C03644=1220.978,171.514,-54.038,-177.762,5.951,148.395
C03645=1220.983,171.266,-54.017,-177.765,5.949,148.395
C03646=1220.988,171.016,-53.994,-177.767,5.948,148.396
C03647=1220.992,170.767,-53.972,-177.770,5.947,148.396
C03648=1220.997,170.518,-53.950,-177.773,5.945,148.397
C03649=1221.001,170.270,-53.928,-177.775,5.943,148.397
C03650=1221.006,170.020,-53.905,-177.777,5.942,148.397
C03651=1221.011,169.771,-53.883,-177.781,5.941,148.398
C03652=1221.015,169.522,-53.861,-177.783,5.940,148.398
C03653=1221.020,169.273,-53.839,-177.785,5.938,148.399
C03654=1221.025,169.025,-53.816,-177.788,5.936,148.399
C03655=1221.029,168.775,-53.794,-177.791,5.936,148.400
C03656=1221.034,168.527,-53.773,-177.793,5.934,148.400
C03657=1221.038,168.277,-53.751,-177.796,5.932,148.400
C03658=1221.043,168.029,-53.729,-177.798,5.931,148.401
C03659=1221.048,167.779,-53.706,-177.801,5.929,148.401
C03660=1221.053,167.530,-53.685,-177.803,5.928,148.402
C03661=1221.057,167.282,-53.662,-177.806,5.927,148.402
C03662=1221.062,167.033,-53.640,-177.809,5.925,148.403
C03663=1221.066,166.784,-53.618,-177.811,5.924,148.403
C03664=1221.071,166.535,-53.596,-177.814,5.922,148.404
C03665=1221.075,166.286,-53.574,-177.816,5.921,148.404
C03666=1221.081,166.037,-53.552,-177.819,5.920,148.405
C03667=1221.085,165.788,-53.530,-177.822,5.918,148.405
C03668=1221.090,165.539,-53.508,-177.824,5.917,148.405
C03669=1221.094,165.290,-53.486,-177.827,5.915,148.406
C03670=1221.099,165.041,-53.465,-177.829,5.915,148.406
C03671=1221.104,164.792,-53.443,-177.832,5.913,148.407
C03672=1221.108,164.543,-53.421,-177.834,5.911,148.407
C03673=1221.113,164.294,-53.399,-177.837,5.910,148.408
C03674=1221.117,164.045,-53.377,-177.840,5.908,148.408
C03675=1221.122,163.796,-53.355,-177.842,5.907,148.408
C03676=1221.127,163.547,-53.333,-177.844,5.906,148.409
C03677=1221.132,163.298,-53.311,-177.848,5.904,148.409
C03678=1221.137,163.049,-53.289,-177.850,5.903,148.410
C03679=1221.141,162.800,-53.267,-177.852,5.901,148.410
C03680=1221.147,162.551,-53.246,-177.855,5.901,148.411
C03681=1221.151,162.301,-53.224,-177.858,5.899,148.411
C03682=1221.156,162.053,-53.203,-177.860,5.897,148.411
C03683=1221.160,161.803,-53.181,-177.863,5.896,148.412
C03684=1221.165,161.555,-53.159,-177.865,5.895,148.412
C03685=1221.170,161.306,-53.137,-177.868,5.894,148.413
C03686=1221.174,161.057,-53.115,-177.870,5.892,148.413
C03687=1221.179,160.808,-53.094,-177.873,5.891,148.414
C03688=1221.183,160.558,-53.072,-177.876,5.889,148.414
C03689=1221.188,160.310,-53.051,-177.878,5.887,148.415
C03690=1221.193,160.061,-53.029,-177.881,5.887,148.415
C03691=1221.198,159.792,-53.006,-177.883,5.885,148.416
C03692=1221.203,159.523,-52.982,-177.887,5.884,148.416
C03693=1221.209,159.254,-52.959,-177.889,5.883,148.417
C03694=1221.213,158.984,-52.936,-177.892,5.881,148.417
C03695=1221.218,158.735,-52.914,-177.894,5.879,148.417
C03696=1221.222,158.487,-52.892,-177.897,5.878,148.418
C03697=1221.227,158.237,-52.870,-177.900,5.877,148.418
C03698=1221.232,157.988,-52.849,-177.902,5.876,148.419
C03699=1221.237,157.740,-52.827,-177.905,5.874,148.419
C03700=1221.241,157.490,-52.805,-177.908,5.872,148.420
C03701=1221.246,157.241,-52.784,-177.910,5.871,148.420
C03702=1221.251,156.992,-52.763,-177.912,5.870,148.421
C03703=1221.255,156.743,-52.741,-177.915,5.869,148.421
C03704=1221.260,156.494,-52.720,-177.918,5.867,148.422
C03705=1221.265,156.245,-52.699,-177.920,5.866,148.422
C03706=1221.270,155.997,-52.677,-177.923,5.865,148.423
C03707=1221.274,155.747,-52.656,-177.925,5.864,148.423
C03708=1221.279,155.498,-52.634,-177.928,5.862,148.423
C03709=1221.284,155.249,-52.612,-177.930,5.861,148.424
C03710=1221.288,155.000,-52.592,-177.933,5.859,148.424
C03711=1221.293,154.751,-52.570,-177.936,5.858,148.425
C03712=1221.298,154.502,-52.549,-177.938,5.857,148.425
C03713=1221.303,154.253,-52.527,-177.941,5.855,148.426
C03714=1221.307,154.003,-52.506,-177.943,5.854,148.426
C03715=1221.312,153.755,-52.484,-177.946,5.853,148.427
C03716=1221.316,153.506,-52.463,-177.948,5.852,148.427
C03717=1221.321,153.256,-52.442,-177.951,5.850,148.427
C03718=1221.326,153.008,-52.420,-177.954,5.849,148.428
C03719=1221.331,152.758,-52.399,-177.956,5.847,148.428
C03720=1221.335,152.510,-52.378,-177.959,5.847,148.429
C03721=1221.339,152.260,-52.357,-177.961,5.845,148.429
C03722=1221.344,152.012,-52.335,-177.964,5.844,148.430
C03723=1221.350,151.762,-52.314,-177.967,5.843,148.430
C03724=1221.354,151.514,-52.293,-177.969,5.842,148.431
C03725=1221.359,151.265,-52.272,-177.971,5.840,148.431
C03726=1221.363,151.015,-52.251,-177.974,5.839,148.432
C03727=1221.368,150.766,-52.229,-177.977,5.837,148.432
C03728=1221.373,150.517,-52.209,-177.979,5.836,148.433
C03729=1221.378,150.269,-52.187,-177.982,5.835,148.433
C03730=1221.383,150.019,-52.166,-177.984,5.834,148.434
C03731=1221.387,149.770,-52.144,-177.987,5.832,148.434
C03732=1221.391,149.521,-52.124,-177.989,5.831,148.435
C03733=1221.397,149.272,-52.103,-177.992,5.830,148.435
C03734=1221.401,149.023,-52.081,-177.995,5.829,148.436
C03735=1221.406,148.774,-52.061,-177.997,5.827,148.436
C03736=1221.410,148.524,-52.039,-178.000,5.827,148.437
C03737=1221.415,148.276,-52.018,-178.003,5.825,148.437
C03738=1221.420,148.027,-51.997,-178.005,5.824,148.437
C03739=1221.425,147.777,-51.976,-178.008,5.822,148.438
C03740=1221.429,147.529,-51.955,-178.010,5.821,148.438
C03741=1221.434,147.280,-51.934,-178.013,5.819,148.439
C03742=1221.439,147.030,-51.913,-178.015,5.819,148.439
C03743=1221.443,146.781,-51.892,-178.018,5.817,148.440
C03744=1221.448,146.532,-51.871,-178.020,5.816,148.440
C03745=1221.453,146.283,-51.850,-178.023,5.815,148.441
C03746=1221.458,146.034,-51.829,-178.025,5.814,148.441
C03747=1221.463,145.785,-51.808,-178.028,5.812,148.442
C03748=1221.467,145.536,-51.787,-178.031,5.811,148.442
C03749=1221.472,145.286,-51.766,-178.034,5.810,148.443
C03750=1221.476,145.037,-51.746,-178.036,5.809,148.443
C03751=1221.481,144.788,-51.725,-178.038,5.807,148.443
C03752=1221.486,144.540,-51.703,-178.041,5.806,148.444
C03753=1221.491,144.291,-51.683,-178.044,5.804,148.444
C03754=1221.496,144.041,-51.662,-178.046,5.804,148.445
C03755=1221.500,143.792,-51.641,-178.049,5.802,148.446
C03756=1221.505,143.543,-51.620,-178.051,5.801,148.446
C03757=1221.510,143.294,-51.600,-178.054,5.800,148.447
C03758=1221.514,143.045,-51.578,-178.056,5.799,148.447
C03759=1221.519,142.796,-51.558,-178.059,5.798,148.448
C03760=1221.524,142.547,-51.537,-178.062,5.796,148.448
C03761=1221.528,142.298,-51.516,-178.064,5.795,148.449
C03762=1221.533,142.048,-51.495,-178.067,5.794,148.449
C03763=1221.538,141.799,-51.475,-178.069,5.793,148.449
C03764=1221.543,141.550,-51.454,-178.072,5.791,148.450
C03765=1221.547,141.301,-51.434,-178.074,5.790,148.450
C03766=1221.553,141.052,-51.413,-178.077,5.789,148.451
C03767=1221.557,140.803,-51.392,-178.080,5.788,148.451
C03768=1221.562,140.554,-51.371,-178.083,5.786,148.452
C03769=1221.567,140.305,-51.351,-178.085,5.785,148.452
C03770=1221.571,140.056,-51.330,-178.087,5.784,148.453
C03771=1221.576,139.807,-51.310,-178.090,5.783,148.453
C03772=1221.581,139.558,-51.289,-178.092,5.782,148.454
C03773=1221.586,139.308,-51.268,-178.095,5.781,148.454
C03774=1221.590,139.059,-51.248,-178.097,5.780,148.455
C03775=1221.595,138.810,-51.227,-178.101,5.778,148.455
C03776=1221.600,138.561,-51.206,-178.103,5.777,148.456
C03777=1221.604,138.312,-51.186,-178.105,5.775,148.456
C03778=1221.609,138.063,-51.165,-178.108,5.775,148.457
C03779=1221.614,137.814,-51.145,-178.110,5.774,148.457
C03780=1221.618,137.565,-51.124,-178.113,5.772,148.458
C03781=1221.623,137.316,-51.103,-178.115,5.771,148.458
C03782=1221.628,137.067,-51.083,-178.119,5.770,148.459
C03783=1221.633,136.818,-51.062,-178.121,5.769,148.459
C03784=1221.638,136.569,-51.042,-178.124,5.767,148.460
C03785=1221.642,136.320,-51.021,-178.126,5.766,148.460
C03786=1221.647,136.070,-51.001,-178.128,5.765,148.461
C03787=1221.652,135.821,-50.981,-178.131,5.764,148.461
C03788=1221.656,135.572,-50.960,-178.133,5.763,148.462
C03789=1221.662,135.323,-50.939,-178.137,5.762,148.462
C03790=1221.666,135.074,-50.919,-178.139,5.761,148.463
C03791=1221.670,134.825,-50.899,-178.141,5.760,148.463
C03792=1221.675,134.575,-50.879,-178.144,5.758,148.464
C03793=1221.680,134.326,-50.858,-178.146,5.757,148.464
C03794=1221.685,134.077,-50.838,-178.149,5.756,148.465
C03795=1221.690,133.808,-50.816,-178.152,5.755,148.465
C03796=1221.695,133.540,-50.794,-178.154,5.753,148.466
C03797=1221.700,133.271,-50.771,-178.157,5.753,148.466
C03798=1221.705,133.002,-50.750,-178.160,5.751,148.467
C03799=1221.710,132.753,-50.729,-178.162,5.750,148.467
C03800=1221.714,132.504,-50.709,-178.165,5.749,148.468
C03801=1221.720,132.255,-50.690,-178.168,5.748,148.468
C03802=1221.725,132.006,-50.669,-178.171,5.746,148.469
C03803=1221.729,131.757,-50.648,-178.173,5.745,148.469
C03804=1221.734,131.508,-50.629,-178.175,5.745,148.470
C03805=1221.738,131.259,-50.608,-178.178,5.743,148.470
C03806=1221.743,131.010,-50.588,-178.181,5.742,148.471
C03807=1221.748,130.760,-50.568,-178.183,5.740,148.471
C03808=1221.753,130.511,-50.547,-178.186,5.740,148.472
C03809=1221.757,130.262,-50.527,-178.188,5.739,148.472
C03810=1221.763,130.013,-50.508,-178.191,5.737,148.473
C03811=1221.767,129.764,-50.487,-178.193,5.736,148.473
C03812=1221.772,129.514,-50.467,-178.197,5.735,148.474
C03813=1221.777,129.265,-50.447,-178.199,5.734,148.474
C03814=1221.781,129.016,-50.426,-178.201,5.733,148.475
C03815=1221.786,128.767,-50.407,-178.204,5.732,148.476
C03816=1221.791,128.518,-50.386,-178.207,5.731,148.476
C03817=1221.796,128.269,-50.367,-178.209,5.730,148.477
C03818=1221.800,128.020,-50.347,-178.212,5.729,148.477
C03819=1221.805,127.771,-50.326,-178.214,5.728,148.478
C03820=1221.810,127.521,-50.306,-178.217,5.726,148.478
C03821=1221.815,127.272,-50.286,-178.219,5.725,148.479
C03822=1221.819,127.023,-50.266,-178.222,5.725,148.479
C03823=1221.824,126.774,-50.246,-178.225,5.723,148.480
C03824=1221.829,126.525,-50.226,-178.227,5.722,148.480
C03825=1221.834,126.276,-50.206,-178.229,5.721,148.481
C03826=1221.838,126.026,-50.186,-178.232,5.720,148.481
C03827=1221.843,125.777,-50.166,-178.235,5.719,148.482
C03828=1221.848,125.528,-50.147,-178.237,5.718,148.482
C03829=1221.853,125.279,-50.127,-178.240,5.716,148.483
C03830=1221.857,125.030,-50.107,-178.242,5.716,148.483
C03831=1221.862,124.780,-50.087,-178.245,5.714,148.484
C03832=1221.866,124.531,-50.067,-178.248,5.713,148.484
C03833=1221.872,124.283,-50.047,-178.250,5.712,148.485
C03834=1221.876,124.034,-50.027,-178.253,5.711,148.485
C03835=1221.881,123.784,-50.007,-178.255,5.710,148.486
C03836=1221.886,123.534,-49.988,-178.258,5.709,148.486
C03837=1221.891,123.286,-49.968,-178.260,5.707,148.487
C03838=1221.896,123.037,-49.948,-178.263,5.707,148.487
C03839=1221.900,122.787,-49.928,-178.265,5.706,148.488
C03840=1221.905,122.538,-49.908,-178.268,5.704,148.489
C03841=1221.910,122.289,-49.889,-178.270,5.703,148.489
C03842=1221.915,122.040,-49.869,-178.273,5.703,148.490
C03843=1221.919,121.791,-49.849,-178.276,5.701,148.490
C03844=1221.924,121.541,-49.829,-178.278,5.700,148.491
C03845=1221.929,121.292,-49.810,-178.281,5.700,148.491
C03846=1221.934,121.043,-49.789,-178.284,5.698,148.492
C03847=1221.939,120.794,-49.770,-178.286,5.697,148.492
C03848=1221.944,120.545,-49.750,-178.288,5.696,148.493
C03849=1221.948,120.296,-49.730,-178.292,5.695,148.493
C03850=1221.953,120.046,-49.710,-178.294,5.694,148.494
C03851=1221.958,119.797,-49.691,-178.296,5.693,148.494
C03852=1221.963,119.548,-49.671,-178.299,5.692,148.495
C03853=1221.968,119.298,-49.652,-178.302,5.691,148.495
C03854=1221.972,119.050,-49.632,-178.304,5.690,148.496
C03855=1221.977,118.801,-49.613,-178.307,5.689,148.496
C03856=1221.982,118.551,-49.593,-178.309,5.688,148.497
C03857=1221.986,118.302,-49.573,-178.312,5.687,148.497
C03858=1221.992,118.053,-49.554,-178.315,5.686,148.498
C03859=1221.996,117.804,-49.534,-178.317,5.685,148.498
C03860=1222.001,117.554,-49.514,-178.320,5.684,148.499
C03861=1222.006,117.306,-49.495,-178.322,5.682,148.500
C03862=1222.010,117.056,-49.476,-178.325,5.682,148.500
C03863=1222.015,116.807,-49.456,-178.327,5.681,148.501
C03864=1222.020,116.558,-49.437,-178.330,5.680,148.501
C03865=1222.025,116.308,-49.417,-178.333,5.679,148.502
C03866=1222.030,116.059,-49.397,-178.335,5.678,148.502
C03867=1222.034,115.811,-49.378,-178.337,5.677,148.503
C03868=1222.039,115.561,-49.358,-178.340,5.675,148.503
C03869=1222.044,115.312,-49.339,-178.343,5.675,148.504
C03870=1222.049,115.063,-49.319,-178.345,5.674,148.504
C03871=1222.054,114.813,-49.300,-178.348,5.672,148.505
C03872=1222.058,114.565,-49.281,-178.351,5.672,148.506
C03873=1222.063,114.315,-49.261,-178.353,5.671,148.506
C03874=1222.068,114.065,-49.242,-178.355,5.670,148.507
C03875=1222.073,113.817,-49.222,-178.358,5.668,148.507
C03876=1222.077,113.567,-49.203,-178.361,5.668,148.508
C03877=1222.083,113.319,-49.184,-178.363,5.667,148.508
C03878=1222.087,113.069,-49.164,-178.366,5.665,148.509
C03879=1222.092,112.819,-49.145,-178.369,5.665,148.509
C03880=1222.097,112.571,-49.126,-178.371,5.664,148.510
C03881=1222.101,112.321,-49.106,-178.373,5.663,148.510
C03882=1222.107,112.072,-49.087,-178.376,5.661,148.511
C03883=1222.111,111.823,-49.067,-178.379,5.661,148.511
C03884=1222.116,111.574,-49.049,-178.381,5.660,148.512
C03885=1222.121,111.325,-49.029,-178.384,5.658,148.512
C03886=1222.126,111.075,-49.009,-178.387,5.658,148.513
C03887=1222.130,110.827,-48.991,-178.389,5.657,148.514
C03888=1222.135,110.577,-48.971,-178.391,5.656,148.514
C03889=1222.141,110.327,-48.952,-178.394,5.654,148.515
C03890=1222.145,110.078,-48.933,-178.397,5.654,148.515
C03891=1222.150,109.829,-48.914,-178.399,5.653,148.516
C03892=1222.155,109.580,-48.894,-178.401,5.652,148.516
C03893=1222.159,109.331,-48.876,-178.404,5.651,148.517
C03894=1222.164,109.082,-48.856,-178.407,5.650,148.517
C03895=1222.169,108.833,-48.837,-178.409,5.649,148.518
C03896=1222.174,108.583,-48.818,-178.412,5.648,148.519
C03897=1222.179,108.334,-48.799,-178.415,5.647,148.519
C03898=1222.183,108.085,-48.780,-178.417,5.646,148.520
C03899=1222.188,107.817,-48.759,-178.420,5.645,148.520
C03900=1222.194,107.548,-48.739,-178.422,5.644,148.521
C03901=1222.199,107.280,-48.718,-178.425,5.643,148.521
C03902=1222.204,107.011,-48.697,-178.428,5.642,148.522
C03903=1222.209,106.762,-48.679,-178.431,5.641,148.523
C03904=1222.214,106.512,-48.660,-178.433,5.640,148.523
C03905=1222.218,106.264,-48.641,-178.436,5.639,148.524
C03906=1222.223,106.014,-48.621,-178.439,5.638,148.524
C03907=1222.228,105.765,-48.603,-178.441,5.637,148.525
C03908=1222.233,105.515,-48.584,-178.443,5.636,148.525
C03909=1222.238,105.267,-48.564,-178.446,5.635,148.526
C03910=1222.242,105.017,-48.545,-178.449,5.634,148.526
C03911=1222.248,104.768,-48.527,-178.451,5.633,148.527
C03912=1222.252,104.519,-48.508,-178.454,5.632,148.527
C03913=1222.257,104.270,-48.488,-178.456,5.632,148.528
C03914=1222.261,104.020,-48.470,-178.459,5.630,148.529
C03915=1222.267,103.771,-48.451,-178.461,5.629,148.529
C03916=1222.271,103.522,-48.432,-178.464,5.629,148.530
C03917=1222.276,103.272,-48.413,-178.466,5.628,148.530
C03918=1222.281,103.024,-48.394,-178.469,5.626,148.531
C03919=1222.286,102.773,-48.375,-178.472,5.626,148.532
C03920=1222.291,102.525,-48.357,-178.474,5.625,148.532
C03921=1222.295,102.275,-48.337,-178.477,5.624,148.533
C03922=1222.300,102.026,-48.319,-178.479,5.624,148.533
C03923=1222.305,101.778,-48.300,-178.482,5.622,148.534
C03924=1222.310,101.527,-48.281,-178.485,5.621,148.534
C03925=1222.315,101.279,-48.263,-178.487,5.620,148.535
C03926=1222.320,101.029,-48.244,-178.489,5.620,148.535
C03927=1222.324,100.780,-48.225,-178.493,5.618,148.536
C03928=1222.330,100.531,-48.206,-178.495,5.617,148.536
C03929=1222.334,100.281,-48.187,-178.497,5.617,148.537
C03930=1222.339,100.033,-48.169,-178.500,5.616,148.538
C03931=1222.344,99.783,-48.150,-178.502,5.615,148.538
C03932=1222.348,99.534,-48.131,-178.505,5.614,148.539
C03933=1222.354,99.285,-48.113,-178.508,5.613,148.539
C03934=1222.358,99.035,-48.094,-178.510,5.612,148.540
C03935=1222.363,98.786,-48.076,-178.513,5.612,148.540
C03936=1222.368,98.537,-48.057,-178.515,5.611,148.541
C03937=1222.372,98.287,-48.038,-178.518,5.609,148.542
C03938=1222.377,98.038,-48.020,-178.521,5.609,148.542
C03939=1222.383,97.789,-48.001,-178.523,5.608,148.543
C03940=1222.387,97.539,-47.982,-178.525,5.607,148.543
C03941=1222.392,97.291,-47.964,-178.528,5.606,148.544
C03942=1222.397,97.041,-47.945,-178.531,5.605,148.545
C03943=1222.402,96.792,-47.927,-178.533,5.604,148.545
C03944=1222.406,96.543,-47.908,-178.536,5.604,148.546
C03945=1222.412,96.293,-47.889,-178.538,5.603,148.546
C03946=1222.416,96.044,-47.870,-178.541,5.602,148.547
C03947=1222.421,95.795,-47.852,-178.544,5.601,148.547
C03948=1222.426,95.546,-47.834,-178.546,5.600,148.548
C03949=1222.430,95.296,-47.815,-178.549,5.599,148.548
C03950=1222.435,95.047,-47.797,-178.551,5.598,148.549
C03951=1222.441,94.798,-47.778,-178.554,5.598,148.550
C03952=1222.445,94.548,-47.759,-178.556,5.596,148.550
C03953=1222.450,94.299,-47.741,-178.559,5.595,148.551
C03954=1222.455,94.050,-47.723,-178.562,5.595,148.551
C03955=1222.460,93.801,-47.704,-178.564,5.594,148.552
C03956=1222.464,93.551,-47.686,-178.566,5.593,148.552
C03957=1222.469,93.302,-47.668,-178.569,5.593,148.553
C03958=1222.474,93.053,-47.650,-178.572,5.591,148.553
C03959=1222.480,92.804,-47.630,-178.574,5.590,148.554
C03960=1222.484,92.554,-47.612,-178.577,5.590,148.555
C03961=1222.489,92.305,-47.594,-178.579,5.589,148.555
C03962=1222.494,92.056,-47.576,-178.582,5.588,148.556
C03963=1222.498,91.807,-47.557,-178.585,5.587,148.557
C03964=1222.503,91.557,-47.538,-178.587,5.586,148.557
C03965=1222.508,91.308,-47.520,-178.590,5.585,148.558
C03966=1222.513,91.059,-47.502,-178.592,5.585,148.558
C03967=1222.518,90.810,-47.484,-178.594,5.584,148.559
C03968=1222.522,90.560,-47.466,-178.597,5.583,148.559
C03969=1222.527,90.311,-47.447,-178.600,5.582,148.560
C03970=1222.533,90.062,-47.429,-178.602,5.581,148.560
C03971=1222.538,89.812,-47.411,-178.605,5.580,148.561
C03972=1222.542,89.563,-47.392,-178.608,5.580,148.562
C03973=1222.547,89.313,-47.374,-178.610,5.579,148.562
C03974=1222.552,89.064,-47.356,-178.612,5.578,148.563
C03975=1222.557,88.815,-47.339,-178.615,5.577,148.563
C03976=1222.561,88.567,-47.320,-178.618,5.576,148.564
C03977=1222.566,88.316,-47.301,-178.620,5.575,148.564
C03978=1222.571,88.067,-47.283,-178.623,5.574,148.565
C03979=1222.576,87.818,-47.265,-178.626,5.574,148.566
C03980=1222.581,87.569,-47.247,-178.628,5.573,148.566
C03981=1222.586,87.320,-47.229,-178.630,5.572,148.567
C03982=1222.590,87.070,-47.211,-178.633,5.572,148.568
C03983=1222.595,86.821,-47.193,-178.636,5.570,148.568
C03984=1222.600,86.571,-47.175,-178.638,5.569,148.569
C03985=1222.605,86.322,-47.157,-178.641,5.569,148.569
C03986=1222.610,86.073,-47.139,-178.644,5.568,148.570
C03987=1222.615,85.824,-47.121,-178.646,5.567,148.570
C03988=1222.619,85.574,-47.102,-178.648,5.567,148.571
C03989=1222.624,85.325,-47.084,-178.651,5.566,148.572
C03990=1222.629,85.076,-47.066,-178.654,5.565,148.572
C03991=1222.635,84.826,-47.048,-178.656,5.564,148.573
C03992=1222.640,84.577,-47.030,-178.659,5.563,148.573
C03993=1222.644,84.328,-47.012,-178.661,5.562,148.574
C03994=1222.649,84.079,-46.994,-178.664,5.562,148.574
C03995=1222.654,83.829,-46.976,-178.666,5.561,148.575
C03996=1222.659,83.580,-46.958,-178.669,5.560,148.576
C03997=1222.663,83.330,-46.940,-178.671,5.560,148.576
C03998=1222.668,83.081,-46.922,-178.674,5.558,148.577
C03999=1222.674,82.831,-46.904,-178.677,5.557,148.577
C04000=1222.679,82.582,-46.886,-178.679,5.557,148.578
C04001=1222.683,82.333,-46.869,-178.682,5.556,148.579
C04002=1222.688,82.084,-46.851,-178.684,5.555,148.579
C04003=1222.693,81.816,-46.831,-178.687,5.555,148.580
C04004=1222.699,81.547,-46.812,-178.690,5.553,148.580
C04005=1222.704,81.279,-46.793,-178.693,5.553,148.581
C04006=1222.709,81.010,-46.773,-178.695,5.552,148.582
C04007=1222.714,80.761,-46.755,-178.698,5.552,148.582
C04008=1222.719,80.512,-46.738,-178.700,5.551,148.583
C04009=1222.723,80.263,-46.720,-178.703,5.549,148.584
C04010=1222.728,80.013,-46.703,-178.706,5.549,148.584
C04011=1222.733,79.764,-46.685,-178.708,5.548,148.585
C04012=1222.738,79.515,-46.667,-178.711,5.547,148.585
C04013=1222.743,79.266,-46.649,-178.713,5.546,148.586
C04014=1222.748,79.016,-46.632,-178.716,5.546,148.587
C04015=1222.753,78.767,-46.614,-178.718,5.545,148.587
C04016=1222.757,78.517,-46.595,-178.721,5.544,148.588
C04017=1222.762,78.268,-46.577,-178.723,5.544,148.588
C04018=1222.767,78.018,-46.561,-178.726,5.543,148.589
C04019=1222.772,77.769,-46.543,-178.729,5.542,148.590
C04020=1222.777,77.520,-46.525,-178.731,5.541,148.590
C04021=1222.781,77.271,-46.507,-178.734,5.540,148.591
C04022=1222.787,77.021,-46.489,-178.736,5.540,148.591
C04023=1222.792,76.772,-46.471,-178.739,5.539,148.592
C04024=1222.796,76.523,-46.454,-178.741,5.538,148.592
C04025=1222.801,76.273,-46.437,-178.744,5.538,148.593
C04026=1222.806,76.024,-46.419,-178.746,5.537,148.594
C04027=1222.811,75.775,-46.401,-178.749,5.536,148.594
C04028=1222.816,75.525,-46.384,-178.751,5.535,148.595
C04029=1222.821,75.276,-46.366,-178.754,5.535,148.596
C04030=1222.825,75.027,-46.348,-178.756,5.534,148.596
C04031=1222.830,74.777,-46.331,-178.760,5.533,148.597
C04032=1222.835,74.528,-46.313,-178.762,5.532,148.597
C04033=1222.840,74.278,-46.296,-178.764,5.531,148.598
C04034=1222.845,74.029,-46.278,-178.767,5.531,148.599
C04035=1222.850,73.780,-46.260,-178.770,5.530,148.599
C04036=1222.855,73.530,-46.243,-178.772,5.529,148.600
C04037=1222.860,73.282,-46.226,-178.774,5.529,148.600
C04038=1222.865,73.032,-46.209,-178.777,5.528,148.601
C04039=1222.870,72.783,-46.191,-178.780,5.528,148.602
C04040=1222.875,72.533,-46.174,-178.782,5.527,148.602
C04041=1222.880,72.284,-46.156,-178.784,5.526,148.603
C04042=1222.884,72.035,-46.139,-178.787,5.525,148.603
C04043=1222.889,71.786,-46.121,-178.790,5.525,148.604
C04044=1222.894,71.536,-46.104,-178.792,5.524,148.605
C04045=1222.899,71.287,-46.086,-178.795,5.523,148.605
C04046=1222.904,71.037,-46.069,-178.798,5.522,148.606
C04047=1222.909,70.788,-46.051,-178.800,5.521,148.606
C04048=1222.914,70.538,-46.034,-178.803,5.521,148.607
C04049=1222.918,70.289,-46.016,-178.806,5.520,148.608
C04050=1222.923,70.039,-45.999,-178.808,5.519,148.608
C04051=1222.929,69.791,-45.982,-178.810,5.519,148.609
C04052=1222.933,69.541,-45.965,-178.813,5.518,148.610
C04053=1222.939,69.292,-45.948,-178.816,5.518,148.610
C04054=1222.943,69.043,-45.930,-178.818,5.517,148.611
C04055=1222.948,68.793,-45.913,-178.820,5.516,148.611
C04056=1222.953,68.544,-45.895,-178.823,5.515,148.612
C04057=1222.957,68.294,-45.878,-178.826,5.515,148.613
C04058=1222.963,68.045,-45.861,-178.828,5.514,148.613
C04059=1222.967,67.795,-45.843,-178.830,5.513,148.614
C04060=1222.973,67.547,-45.827,-178.833,5.513,148.614
C04061=1222.977,67.297,-45.809,-178.836,5.512,148.615
C04062=1222.982,67.048,-45.792,-178.838,5.512,148.616
C04063=1222.987,66.798,-45.775,-178.841,5.511,148.616
C04064=1222.992,66.549,-45.757,-178.843,5.510,148.617
C04065=1222.997,66.299,-45.740,-178.846,5.509,148.617
C04066=1223.002,66.050,-45.723,-178.849,5.508,148.618
C04067=1223.007,65.802,-45.706,-178.852,5.508,148.619
C04068=1223.012,65.552,-45.689,-178.854,5.507,148.619
C04069=1223.016,65.302,-45.672,-178.856,5.506,148.620
C04070=1223.021,65.052,-45.655,-178.859,5.505,148.621
C04071=1223.026,64.804,-45.637,-178.862,5.505,148.621
C04072=1223.031,64.554,-45.620,-178.864,5.504,148.622
C04073=1223.037,64.305,-45.603,-178.867,5.504,148.623
C04074=1223.041,64.055,-45.587,-178.869,5.503,148.623
C04075=1223.046,63.806,-45.569,-178.872,5.502,148.624
C04076=1223.051,63.557,-45.552,-178.874,5.502,148.624
C04077=1223.056,63.307,-45.535,-178.877,5.501,148.625
C04078=1223.060,63.057,-45.518,-178.879,5.501,148.626
C04079=1223.066,62.809,-45.500,-178.882,5.500,148.626
C04080=1223.070,62.559,-45.484,-178.884,5.499,148.627
C04081=1223.075,62.310,-45.466,-178.887,5.498,148.627
C04082=1223.080,62.060,-45.450,-178.890,5.498,148.628
C04083=1223.086,61.811,-45.433,-178.892,5.497,148.629
C04084=1223.090,61.561,-45.416,-178.894,5.496,148.629
C04085=1223.094,61.313,-45.399,-178.897,5.496,148.630
C04086=1223.100,61.063,-45.381,-178.900,5.495,148.630
C04087=1223.104,60.813,-45.365,-178.902,5.495,148.631
C04088=1223.110,60.564,-45.348,-178.905,5.494,148.632
C04089=1223.114,60.315,-45.331,-178.907,5.493,148.632
C04090=1223.120,60.065,-45.314,-178.910,5.493,148.633
C04091=1223.124,59.815,-45.297,-178.912,5.492,148.634
C04092=1223.130,59.566,-45.280,-178.915,5.491,148.634
C04093=1223.134,59.317,-45.264,-178.917,5.491,148.635
C04094=1223.139,59.068,-45.246,-178.920,5.490,148.636
C04095=1223.144,58.818,-45.229,-178.922,5.489,148.636
C04096=1223.149,58.569,-45.213,-178.925,5.489,148.637
C04097=1223.154,58.320,-45.196,-178.928,5.488,148.637
C04098=1223.159,58.070,-45.179,-178.930,5.488,148.638
C04099=1223.164,57.821,-45.163,-178.933,5.487,148.639
C04100=1223.169,57.572,-45.145,-178.935,5.487,148.639
C04101=1223.173,57.322,-45.129,-178.938,5.486,148.640
C04102=1223.178,57.073,-45.112,-178.940,5.485,148.640
C04103=1223.184,56.824,-45.095,-178.943,5.484,148.641
C04104=1223.188,56.574,-45.078,-178.945,5.484,148.642
C04105=1223.193,56.325,-45.062,-178.948,5.483,148.642
C04106=1223.198,56.075,-45.045,-178.950,5.482,148.643
C04107=1223.203,55.807,-45.027,-178.953,5.482,148.644
C04108=1223.209,55.538,-45.009,-178.956,5.482,148.644
C04109=1223.214,55.270,-44.991,-178.959,5.481,148.645
C04110=1223.219,55.002,-44.973,-178.962,5.480,148.646
C04111=1223.225,54.752,-44.956,-178.965,5.479,148.646
C04112=1223.229,54.502,-44.939,-178.967,5.478,148.647
C04113=1223.234,54.254,-44.923,-178.969,5.478,148.648
C04114=1223.239,54.004,-44.906,-178.971,5.478,148.648
C04115=1223.244,53.754,-44.890,-178.974,5.477,148.649
C04116=1223.249,53.505,-44.874,-178.977,5.477,148.650
C04117=1223.254,53.255,-44.857,-178.979,5.476,148.650
C04118=1223.259,53.006,-44.840,-178.981,5.475,148.651
C04119=1223.264,52.757,-44.823,-178.984,5.475,148.651
C04120=1223.268,52.507,-44.807,-178.987,5.474,148.652
C04121=1223.273,52.259,-44.790,-178.989,5.474,148.653
C04122=1223.279,52.008,-44.774,-178.992,5.473,148.653
C04123=1223.283,51.759,-44.757,-178.995,5.472,148.654
C04124=1223.289,51.510,-44.741,-178.997,5.472,148.654
C04125=1223.293,51.260,-44.724,-178.999,5.471,148.655
C04126=1223.298,51.011,-44.707,-179.002,5.470,148.656
C04127=1223.303,50.762,-44.691,-179.005,5.470,148.656
C04128=1223.308,50.512,-44.675,-179.007,5.469,148.657
C04129=1223.313,50.263,-44.658,-179.010,5.469,148.658
C04130=1223.318,50.014,-44.642,-179.013,5.468,148.658
C04131=1223.322,49.764,-44.625,-179.015,5.467,148.659
C04132=1223.328,49.514,-44.609,-179.017,5.467,148.660
C04133=1223.333,49.265,-44.592,-179.020,5.466,148.660
C04134=1223.338,49.016,-44.576,-179.023,5.466,148.661
C04135=1223.342,48.767,-44.559,-179.025,5.465,148.662
C04136=1223.347,48.516,-44.543,-179.028,5.464,148.662
C04137=1223.352,48.268,-44.527,-179.031,5.464,148.663
C04138=1223.357,48.018,-44.510,-179.033,5.463,148.663
C04139=1223.363,47.768,-44.494,-179.035,5.462,148.664
C04140=1223.367,47.519,-44.477,-179.037,5.463,148.665
C04141=1223.372,47.270,-44.461,-179.040,5.462,148.665
C04142=1223.377,47.020,-44.445,-179.043,5.461,148.666
C04143=1223.382,46.771,-44.429,-179.045,5.461,148.667
C04144=1223.387,46.522,-44.412,-179.048,5.460,148.667
C04145=1223.392,46.272,-44.396,-179.051,5.460,148.668
C04146=1223.397,46.023,-44.379,-179.053,5.459,148.669
C04147=1223.402,45.773,-44.363,-179.055,5.458,148.669
C04148=1223.407,45.524,-44.347,-179.058,5.458,148.670
C04149=1223.412,45.274,-44.330,-179.061,5.457,148.671
C04150=1223.417,45.025,-44.315,-179.063,5.457,148.671
C04151=1223.422,44.775,-44.298,-179.066,5.456,148.672
C04152=1223.427,44.527,-44.282,-179.069,5.456,148.673
C04153=1223.431,44.276,-44.266,-179.071,5.455,148.673
C04154=1223.436,44.028,-44.250,-179.073,5.454,148.674
C04155=1223.441,43.778,-44.234,-179.076,5.454,148.674
C04156=1223.446,43.529,-44.217,-179.078,5.454,148.675
C04157=1223.451,43.279,-44.201,-179.081,5.453,148.676
C04158=1223.456,43.030,-44.185,-179.083,5.453,148.676
C04159=1223.461,42.780,-44.168,-179.086,5.452,148.677
C04160=1223.466,42.531,-44.153,-179.089,5.452,148.678
C04161=1223.471,42.282,-44.136,-179.091,5.451,148.678
C04162=1223.476,42.032,-44.121,-179.093,5.450,148.679
C04163=1223.480,41.783,-44.104,-179.096,5.450,148.679
C04164=1223.486,41.533,-44.088,-179.099,5.449,148.680
C04165=1223.491,41.283,-44.072,-179.101,5.448,148.681
C04166=1223.496,41.034,-44.056,-179.104,5.448,148.682
C04167=1223.500,40.784,-44.040,-179.107,5.447,148.682
C04168=1223.506,40.536,-44.024,-179.109,5.447,148.683
C04169=1223.511,40.286,-44.008,-179.111,5.447,148.684
C04170=1223.515,40.037,-43.991,-179.113,5.446,148.684
C04171=1223.521,39.787,-43.976,-179.116,5.446,148.685
C04172=1223.525,39.538,-43.959,-179.119,5.445,148.685
C04173=1223.531,39.288,-43.944,-179.121,5.444,148.686
C04174=1223.535,39.038,-43.928,-179.124,5.444,148.687
C04175=1223.541,38.789,-43.911,-179.127,5.443,148.687
C04176=1223.545,38.539,-43.895,-179.129,5.443,148.688
C04177=1223.550,38.291,-43.879,-179.132,5.442,148.689
C04178=1223.556,38.041,-43.864,-179.135,5.442,148.689
C04179=1223.561,37.791,-43.848,-179.137,5.441,148.690
C04180=1223.566,37.542,-43.831,-179.139,5.441,148.691
C04181=1223.570,37.292,-43.815,-179.141,5.440,148.691
C04182=1223.575,37.043,-43.800,-179.144,5.440,148.692
C04183=1223.580,36.794,-43.784,-179.147,5.439,148.693
C04184=1223.585,36.544,-43.768,-179.149,5.439,148.693
C04185=1223.590,36.295,-43.752,-179.152,5.438,148.694
C04186=1223.595,36.045,-43.736,-179.155,5.438,148.695
C04187=1223.600,35.796,-43.720,-179.157,5.437,148.695
C04188=1223.606,35.546,-43.705,-179.159,5.436,148.696
C04189=1223.610,35.297,-43.689,-179.162,5.436,148.696
C04190=1223.615,35.048,-43.673,-179.164,5.436,148.697
C04191=1223.620,34.799,-43.657,-179.167,5.435,148.698
C04192=1223.625,34.548,-43.641,-179.169,5.435,148.698
C04193=1223.630,34.299,-43.626,-179.172,5.434,148.699
C04194=1223.635,34.050,-43.609,-179.175,5.434,148.700
C04195=1223.639,33.800,-43.594,-179.177,5.433,148.700
C04196=1223.645,33.551,-43.579,-179.180,5.433,148.701
C04197=1223.650,33.301,-43.563,-179.183,5.432,148.702
C04198=1223.655,33.052,-43.546,-179.184,5.432,148.702
C04199=1223.660,32.803,-43.531,-179.187,5.431,148.703
C04200=1223.664,32.553,-43.515,-179.189,5.431,148.704
C04201=1223.670,32.304,-43.500,-179.192,5.430,148.704
C04202=1223.675,32.054,-43.484,-179.195,5.430,148.705
C04203=1223.680,31.804,-43.468,-179.197,5.429,148.706
C04204=1223.685,31.555,-43.452,-179.200,5.429,148.706
C04205=1223.689,31.306,-43.437,-179.203,5.428,148.707
C04206=1223.694,31.056,-43.421,-179.205,5.428,148.708
C04207=1223.700,30.807,-43.405,-179.207,5.428,148.708
C04208=1223.705,30.557,-43.390,-179.210,5.427,148.709
C04209=1223.710,30.308,-43.375,-179.212,5.426,148.709
C04210=1223.714,30.058,-43.359,-179.215,5.426,148.710
C04211=1223.720,29.790,-43.342,-179.218,5.426,148.711
C04212=1223.726,29.521,-43.325,-179.221,5.425,148.712
C04213=1223.730,29.253,-43.308,-179.223,5.425,148.712
C04214=1223.736,28.984,-43.291,-179.226,5.424,148.713
C04215=1223.741,28.734,-43.275,-179.229,5.424,148.714
C04216=1223.745,28.485,-43.260,-179.231,5.423,148.714
C04217=1223.751,28.236,-43.245,-179.234,5.422,148.715
C04218=1223.756,27.986,-43.229,-179.236,5.423,148.716
C04219=1223.761,27.736,-43.213,-179.239,5.422,148.716
C04220=1223.766,27.487,-43.198,-179.241,5.421,148.717
C04221=1223.771,27.238,-43.183,-179.243,5.421,148.718
C04222=1223.776,26.988,-43.167,-179.246,5.420,148.718
C04223=1223.780,26.739,-43.152,-179.249,5.420,148.719
C04224=1223.786,26.489,-43.136,-179.251,5.419,148.720
C04225=1223.791,26.240,-43.121,-179.253,5.419,148.720
C04226=1223.796,25.991,-43.106,-179.256,5.419,148.721
C04227=1223.801,25.741,-43.090,-179.259,5.418,148.722
C04228=1223.805,25.492,-43.075,-179.261,5.418,148.722
C04229=1223.811,25.242,-43.059,-179.264,5.417,148.723
C04230=1223.816,24.993,-43.044,-179.267,5.417,148.724
C04231=1223.820,24.743,-43.028,-179.269,5.416,148.724
C04232=1223.826,24.493,-43.013,-179.271,5.416,148.725
C04233=1223.830,24.244,-42.998,-179.274,5.416,148.726
C04234=1223.836,23.994,-42.983,-179.276,5.415,148.726
C04235=1223.841,23.745,-42.967,-179.279,5.414,148.727
C04236=1223.845,23.495,-42.952,-179.281,5.414,148.728
C04237=1223.851,23.246,-42.936,-179.284,5.413,148.728
C04238=1223.855,22.997,-42.921,-179.286,5.414,148.729
C04239=1223.861,22.747,-42.906,-179.289,5.413,148.730
C04240=1223.865,22.498,-42.891,-179.291,5.413,148.730
C04241=1223.870,22.248,-42.875,-179.294,5.412,148.731
C04242=1223.876,21.998,-42.860,-179.297,5.411,148.732
C04243=1223.880,21.749,-42.845,-179.299,5.411,148.732
C04244=1223.886,21.500,-42.829,-179.301,5.411,148.733
C04245=1223.890,21.251,-42.814,-179.304,5.411,148.734
C04246=1223.896,21.001,-42.799,-179.307,5.410,148.734
C04247=1223.900,20.751,-42.784,-179.309,5.410,148.735
C04248=1223.906,20.501,-42.768,-179.312,5.409,148.736
C04249=1223.910,20.252,-42.753,-179.314,5.408,148.736
C04250=1223.916,20.003,-42.738,-179.316,5.408,148.737
C04251=1223.920,19.754,-42.723,-179.319,5.408,148.738
C04252=1223.926,19.504,-42.708,-179.322,5.407,148.738
C04253=1223.930,19.254,-42.693,-179.324,5.407,148.739
C04254=1223.935,19.005,-42.677,-179.327,5.406,148.740
C04255=1223.940,18.755,-42.662,-179.329,5.406,148.740
C04256=1223.946,18.505,-42.647,-179.332,5.406,148.741
C04257=1223.950,18.256,-42.632,-179.334,5.405,148.742
C04258=1223.956,18.007,-42.617,-179.337,5.405,148.742
C04259=1223.961,17.757,-42.602,-179.339,5.404,148.743
C04260=1223.965,17.508,-42.587,-179.342,5.404,148.744
C04261=1223.970,17.258,-42.571,-179.344,5.404,148.744
C04262=1223.975,17.009,-42.556,-179.347,5.404,148.745
C04263=1223.980,16.759,-42.541,-179.349,5.403,148.746
C04264=1223.985,16.510,-42.526,-179.352,5.403,148.746
C04265=1223.991,16.260,-42.511,-179.355,5.402,148.747
C04266=1223.995,16.011,-42.497,-179.357,5.401,148.748
C04267=1224.000,15.762,-42.482,-179.359,5.401,148.748
C04268=1224.006,15.512,-42.466,-179.362,5.401,148.749
C04269=1224.010,15.263,-42.452,-179.364,5.400,148.750
C04270=1224.016,15.013,-42.436,-179.367,5.400,148.750
C04271=1224.021,14.763,-42.422,-179.370,5.399,148.751
C04272=1224.025,14.514,-42.407,-179.372,5.400,148.752
C04273=1224.030,14.264,-42.391,-179.374,5.399,148.752
C04274=1224.035,14.014,-42.377,-179.377,5.398,148.753
C04275=1224.040,13.765,-42.362,-179.380,5.398,148.754
C04276=1224.046,13.515,-42.347,-179.382,5.397,148.754
C04277=1224.050,13.266,-42.332,-179.384,5.398,148.755
C04278=1224.056,13.016,-42.317,-179.387,5.397,148.756
C04279=1224.061,12.767,-42.302,-179.390,5.397,148.756
C04280=1224.065,12.518,-42.287,-179.392,5.396,148.757
C04281=1224.071,12.268,-42.272,-179.395,5.396,148.758
C04282=1224.076,12.019,-42.257,-179.397,5.396,148.759
C04283=1224.080,11.769,-42.243,-179.400,5.395,148.759
C04284=1224.086,11.520,-42.227,-179.402,5.395,148.760
C04285=1224.091,11.270,-42.213,-179.405,5.394,148.761
C04286=1224.095,11.021,-42.198,-179.408,5.394,148.761
C04287=1224.100,10.771,-42.184,-179.409,5.394,148.762
C04288=1224.106,10.522,-42.168,-179.412,5.393,148.762
C04289=1224.111,10.272,-42.154,-179.415,5.393,148.763
C04290=1224.115,10.023,-42.139,-179.417,5.392,148.764
C04291=1224.121,9.773,-42.124,-179.420,5.392,148.764
C04292=1224.126,9.523,-42.110,-179.422,5.392,148.765
C04293=1224.131,9.274,-42.095,-179.425,5.391,148.766
C04294=1224.136,9.025,-42.080,-179.427,5.391,148.766
C04295=1224.141,8.775,-42.065,-179.430,5.390,148.767
C04296=1224.146,8.525,-42.051,-179.432,5.391,148.768
C04297=1224.151,8.276,-42.036,-179.435,5.390,148.769
C04298=1224.156,8.027,-42.021,-179.437,5.389,148.769
C04299=1224.161,7.777,-42.006,-179.440,5.389,148.770
C04300=1224.166,7.528,-41.991,-179.443,5.388,148.771
C04301=1224.171,7.278,-41.977,-179.445,5.389,148.771
C04302=1224.176,7.029,-41.962,-179.447,5.388,148.772
C04303=1224.181,6.779,-41.948,-179.450,5.388,148.773
C04304=1224.186,6.529,-41.933,-179.453,5.387,148.773
C04305=1224.191,6.280,-41.918,-179.455,5.387,148.774
C04306=1224.196,6.030,-41.904,-179.457,5.387,148.775
C04307=1224.201,5.781,-41.889,-179.460,5.386,148.775
C04308=1224.205,5.531,-41.874,-179.463,5.386,148.776
C04309=1224.210,5.282,-41.860,-179.465,5.385,148.777
C04310=1224.217,5.032,-41.846,-179.467,5.386,148.777
C04311=1224.221,4.783,-41.831,-179.470,5.385,148.778
C04312=1224.226,4.534,-41.816,-179.473,5.385,148.779
C04313=1224.231,4.284,-41.802,-179.475,5.384,148.780
C04314=1224.236,4.034,-41.788,-179.477,5.384,148.780
C04315=1224.241,3.765,-41.772,-179.480,5.384,148.781
C04316=1224.247,3.496,-41.756,-179.483,5.383,148.782
C04317=1224.252,3.228,-41.740,-179.485,5.383,148.782
C04318=1224.258,2.958,-41.725,-179.488,5.382,148.783
C04319=1224.262,2.709,-41.710,-179.491,5.382,148.784
C04320=1224.267,2.459,-41.696,-179.493,5.382,148.784
C04321=1224.273,2.210,-41.682,-179.495,5.381,148.785
C04322=1224.279,1.960,-41.667,-179.498,5.381,148.786
C04323=1224.283,1.711,-41.652,-179.501,5.380,148.786
C04324=1224.288,1.461,-41.638,-179.503,5.381,148.787
C04325=1224.293,1.212,-41.624,-179.505,5.380,148.788
C04326=1224.298,0.962,-41.609,-179.508,5.380,148.788
C04327=1224.303,0.712,-41.595,-179.511,5.379,148.789
C04328=1224.308,0.463,-41.581,-179.513,5.379,148.790
C04329=1224.313,0.214,-41.566,-179.515,5.379,148.791
C04330=1224.318,-0.035,-41.552,-179.518,5.378,148.791
C04331=1224.323,-0.285,-41.537,-179.521,5.378,148.792
C04332=1224.328,-0.535,-41.523,-179.523,5.378,148.793
C04333=1224.333,-0.785,-41.509,-179.525,5.378,148.793
C04334=1224.338,-1.034,-41.495,-179.528,5.377,148.794
C04335=1224.344,-1.283,-41.481,-179.531,5.377,148.795
C04336=1224.349,-1.533,-41.466,-179.533,5.377,148.795
C04337=1224.353,-1.782,-41.451,-179.535,5.376,148.796
C04338=1224.358,-2.032,-41.437,-179.538,5.376,148.797
C04339=1224.363,-2.282,-41.423,-179.541,5.375,148.797
C04340=1224.368,-2.531,-41.409,-179.543,5.376,148.798
C04341=1224.374,-2.780,-41.395,-179.545,5.375,148.799
C04342=1224.379,-3.030,-41.380,-179.548,5.375,148.800
C04343=1224.384,-3.280,-41.366,-179.551,5.374,148.800
C04344=1224.388,-3.529,-41.352,-179.553,5.374,148.801
C04345=1224.393,-3.779,-41.338,-179.556,5.374,148.802
C04346=1224.399,-4.028,-41.324,-179.558,5.373,148.802
C04347=1224.404,-4.278,-41.309,-179.561,5.373,148.803
C04348=1224.409,-4.528,-41.295,-179.563,5.373,148.804
C04349=1224.414,-4.777,-41.281,-179.566,5.373,148.804
C04350=1224.419,-5.027,-41.267,-179.568,5.372,148.805
C04351=1224.424,-5.276,-41.253,-179.571,5.372,148.806
C04352=1224.429,-5.526,-41.238,-179.573,5.372,148.806
C04353=1224.434,-5.775,-41.224,-179.576,5.371,148.807
C04354=1224.439,-6.025,-41.210,-179.578,5.371,148.808
C04355=1224.444,-6.275,-41.196,-179.580,5.371,148.809
C04356=1224.450,-6.524,-41.182,-179.583,5.371,148.809
C04357=1224.455,-6.774,-41.167,-179.586,5.370,148.810
C04358=1224.459,-7.023,-41.154,-179.588,5.370,148.811
C04359=1224.464,-7.273,-41.139,-179.590,5.370,148.811
C04360=1224.469,-7.522,-41.126,-179.593,5.369,148.812
C04361=1224.474,-7.771,-41.111,-179.596,5.369,148.813
C04362=1224.480,-8.022,-41.098,-179.597,5.369,148.813
C04363=1224.485,-8.271,-41.083,-179.600,5.368,148.814
C04364=1224.490,-8.520,-41.070,-179.603,5.368,148.814
C04365=1224.495,-8.770,-41.055,-179.605,5.367,148.815
C04366=1224.499,-9.020,-41.042,-179.607,5.368,148.816
C04367=1224.504,-9.269,-41.027,-179.610,5.367,148.817
C04368=1224.510,-9.518,-41.013,-179.613,5.367,148.817
C04369=1224.515,-9.768,-40.999,-179.615,5.367,148.818
C04370=1224.520,-10.018,-40.986,-179.617,5.366,148.819
C04371=1224.526,-10.267,-40.972,-179.620,5.366,148.819
C04372=1224.530,-10.517,-40.958,-179.623,5.365,148.820
C04373=1224.535,-10.766,-40.944,-179.625,5.366,148.821
C04374=1224.540,-11.016,-40.929,-179.627,5.365,148.821
C04375=1224.546,-11.266,-40.916,-179.630,5.365,148.822
C04376=1224.551,-11.515,-40.902,-179.632,5.365,148.823
C04377=1224.555,-11.765,-40.888,-179.635,5.364,148.823
C04378=1224.560,-12.014,-40.874,-179.637,5.364,148.824
C04379=1224.565,-12.264,-40.860,-179.640,5.363,148.825
C04380=1224.571,-12.514,-40.846,-179.642,5.364,148.826
C04381=1224.576,-12.763,-40.833,-179.645,5.363,148.826
C04382=1224.580,-13.012,-40.819,-179.648,5.363,148.827
C04383=1224.585,-13.262,-40.805,-179.650,5.363,148.828
C04384=1224.591,-13.512,-40.791,-179.652,5.362,148.828
C04385=1224.596,-13.761,-40.777,-179.655,5.362,148.829
C04386=1224.600,-14.011,-40.763,-179.657,5.362,148.830
C04387=1224.606,-14.260,-40.750,-179.660,5.362,148.830
C04388=1224.611,-14.510,-40.736,-179.662,5.361,148.831
C04389=1224.616,-14.760,-40.722,-179.665,5.361,148.832
C04390=1224.621,-15.009,-40.708,-179.667,5.361,148.833
C04391=1224.626,-15.259,-40.695,-179.670,5.361,148.833
C04392=1224.631,-15.509,-40.681,-179.672,5.360,148.834
C04393=1224.637,-15.758,-40.667,-179.674,5.360,148.835
C04394=1224.641,-16.008,-40.654,-179.677,5.360,148.835
C04395=1224.647,-16.257,-40.640,-179.680,5.359,148.836
C04396=1224.652,-16.506,-40.625,-179.682,5.360,148.837
C04397=1224.656,-16.756,-40.612,-179.684,5.359,148.837
C04398=1224.662,-17.005,-40.599,-179.687,5.359,148.838
C04399=1224.667,-17.256,-40.585,-179.689,5.359,148.839
C04400=1224.672,-17.504,-40.572,-179.692,5.358,148.839
C04401=1224.677,-17.754,-40.557,-179.695,5.358,148.840
C04402=1224.682,-18.004,-40.544,-179.697,5.357,148.841
C04403=1224.687,-18.253,-40.531,-179.699,5.358,148.842
C04404=1224.692,-18.503,-40.517,-179.702,5.357,148.842
C04405=1224.698,-18.752,-40.503,-179.705,5.357,148.843
C04406=1224.702,-19.002,-40.489,-179.707,5.357,148.844
C04407=1224.707,-19.252,-40.476,-179.709,5.356,148.844
C04408=1224.713,-19.501,-40.462,-179.712,5.356,148.845
C04409=1224.717,-19.751,-40.449,-179.714,5.356,148.846
C04410=1224.723,-20.000,-40.435,-179.717,5.356,148.846
C04411=1224.728,-20.251,-40.421,-179.719,5.355,148.847
C04412=1224.733,-20.499,-40.408,-179.721,5.356,148.848
C04413=1224.738,-20.750,-40.395,-179.724,5.355,148.848
C04414=1224.742,-20.999,-40.381,-179.727,5.355,148.849
C04415=1224.748,-21.249,-40.368,-179.729,5.355,148.850
C04416=1224.753,-21.498,-40.353,-179.732,5.354,148.851
C04417=1224.758,-21.748,-40.341,-179.734,5.354,148.851
C04418=1224.763,-21.997,-40.327,-179.736,5.354,148.852
C04419=1224.769,-22.266,-40.313,-179.739,5.354,148.853
C04420=1224.774,-22.536,-40.298,-179.742,5.354,148.854
C04421=1224.780,-22.805,-40.283,-179.745,5.353,148.854
C04422=1224.785,-23.075,-40.268,-179.747,5.353,148.855
C04423=1224.790,-23.324,-40.256,-179.749,5.353,148.856
C04424=1224.796,-23.574,-40.242,-179.752,5.352,148.856
C04425=1224.800,-23.823,-40.229,-179.755,5.352,148.857
C04426=1224.806,-24.073,-40.215,-179.757,5.352,148.858
C04427=1224.810,-24.322,-40.202,-179.760,5.352,148.858
C04428=1224.816,-24.572,-40.188,-179.762,5.351,148.859
C04429=1224.821,-24.822,-40.176,-179.764,5.351,148.860
C04430=1224.826,-25.071,-40.161,-179.767,5.351,148.861
C04431=1224.831,-25.321,-40.149,-179.770,5.350,148.861
C04432=1224.836,-25.570,-40.135,-179.772,5.351,148.862
C04433=1224.841,-25.820,-40.122,-179.774,5.350,148.863
C04434=1224.846,-26.070,-40.108,-179.777,5.350,148.863
C04435=1224.851,-26.319,-40.095,-179.779,5.350,148.864
C04436=1224.856,-26.569,-40.082,-179.782,5.350,148.865
C04437=1224.861,-26.818,-40.069,-179.784,5.349,148.865
C04438=1224.866,-27.068,-40.055,-179.786,5.349,148.866
C04439=1224.872,-27.317,-40.042,-179.789,5.349,148.867
C04440=1224.877,-27.568,-40.029,-179.792,5.348,148.868
C04441=1224.882,-27.816,-40.015,-179.794,5.349,148.868
C04442=1224.887,-28.067,-40.002,-179.797,5.348,148.869
C04443=1224.892,-28.316,-39.989,-179.799,5.349,148.870
C04444=1224.896,-28.566,-39.976,-179.801,5.348,148.870
C04445=1224.902,-28.815,-39.962,-179.804,5.348,148.871
C04446=1224.907,-29.064,-39.950,-179.806,5.348,148.872
C04447=1224.912,-29.315,-39.936,-179.809,5.347,148.872
C04448=1224.918,-29.564,-39.923,-179.811,5.347,148.873
C04449=1224.923,-29.814,-39.909,-179.813,5.347,148.874
C04450=1224.928,-30.063,-39.897,-179.816,5.347,148.874
C04451=1224.932,-30.313,-39.884,-179.819,5.346,148.875
C04452=1224.938,-30.563,-39.870,-179.821,5.347,148.876
C04453=1224.943,-30.811,-39.857,-179.824,5.346,148.877
C04454=1224.948,-31.062,-39.843,-179.826,5.346,148.877
C04455=1224.953,-31.311,-39.831,-179.828,5.346,148.878
C04456=1224.958,-31.561,-39.818,-179.831,5.345,148.879
C04457=1224.964,-31.811,-39.805,-179.834,5.345,148.879
C04458=1224.968,-32.059,-39.791,-179.836,5.345,148.880
C04459=1224.973,-32.309,-39.778,-179.838,5.345,148.881
C04460=1224.979,-32.559,-39.765,-179.840,5.345,148.881
C04461=1224.983,-32.809,-39.752,-179.843,5.345,148.882
C04462=1224.988,-33.058,-39.740,-179.846,5.344,148.883
C04463=1224.994,-33.308,-39.726,-179.848,5.344,148.884
C04464=1224.999,-33.558,-39.714,-179.850,5.344,148.884
C04465=1225.004,-33.807,-39.700,-179.853,5.343,148.885
C04466=1225.009,-34.057,-39.687,-179.855,5.344,148.886
C04467=1225.014,-34.306,-39.674,-179.858,5.343,148.886
C04468=1225.019,-34.556,-39.661,-179.861,5.343,148.887
C04469=1225.024,-34.806,-39.648,-179.863,5.343,148.888
C04470=1225.030,-35.055,-39.635,-179.865,5.343,148.888
C04471=1225.035,-35.305,-39.623,-179.867,5.343,148.889
C04472=1225.040,-35.555,-39.609,-179.870,5.342,148.890
C04473=1225.045,-35.804,-39.597,-179.873,5.342,148.891
C04474=1225.050,-36.054,-39.584,-179.875,5.342,148.891
C04475=1225.055,-36.304,-39.571,-179.877,5.342,148.892
C04476=1225.061,-36.553,-39.558,-179.880,5.341,148.893
C04477=1225.066,-36.803,-39.545,-179.882,5.342,148.893
C04478=1225.070,-37.052,-39.531,-179.885,5.341,148.894
C04479=1225.076,-37.302,-39.518,-179.887,5.341,148.895
C04480=1225.081,-37.551,-39.506,-179.890,5.341,148.895
C04481=1225.085,-37.801,-39.493,-179.892,5.340,148.896
C04482=1225.091,-38.050,-39.480,-179.894,5.341,148.897
C04483=1225.096,-38.300,-39.468,-179.897,5.340,148.898
C04484=1225.101,-38.550,-39.454,-179.900,5.340,148.898
C04485=1225.106,-38.800,-39.442,-179.902,5.340,148.899
C04486=1225.111,-39.049,-39.429,-179.904,5.340,148.900
C04487=1225.116,-39.299,-39.416,-179.906,5.340,148.900
C04488=1225.122,-39.549,-39.403,-179.909,5.339,148.901
C04489=1225.127,-39.798,-39.391,-179.912,5.339,148.902
C04490=1225.132,-40.047,-39.378,-179.914,5.339,148.902
C04491=1225.137,-40.297,-39.365,-179.917,5.339,148.903
C04492=1225.142,-40.547,-39.353,-179.919,5.338,148.904
C04493=1225.148,-40.796,-39.339,-179.921,5.339,148.905
C04494=1225.152,-41.046,-39.326,-179.924,5.338,148.905
C04495=1225.157,-41.296,-39.314,-179.926,5.338,148.906
C04496=1225.162,-41.545,-39.301,-179.929,5.338,148.907
C04497=1225.168,-41.794,-39.289,-179.931,5.337,148.907
C04498=1225.172,-42.044,-39.276,-179.933,5.338,148.908
C04499=1225.177,-42.294,-39.264,-179.936,5.337,148.909
C04500=1225.183,-42.544,-39.251,-179.938,5.338,148.909
C04501=1225.188,-42.793,-39.238,-179.941,5.337,148.910
C04502=1225.193,-43.043,-39.225,-179.944,5.337,148.911
C04503=1225.198,-43.293,-39.212,-179.946,5.337,148.912
C04504=1225.203,-43.542,-39.200,-179.948,5.336,148.912
C04505=1225.209,-43.792,-39.188,-179.950,5.337,148.913
C04506=1225.213,-44.042,-39.175,-179.953,5.336,148.914
C04507=1225.218,-44.291,-39.162,-179.956,5.336,148.914
C04508=1225.224,-44.541,-39.149,-179.958,5.336,148.915
C04509=1225.229,-44.790,-39.136,-179.960,5.336,148.916
C04510=1225.234,-45.040,-39.124,-179.963,5.336,148.916
C04511=1225.239,-45.290,-39.112,-179.965,5.336,148.917
C04512=1225.244,-45.539,-39.099,-179.968,5.335,148.918
C04513=1225.249,-45.789,-39.086,-179.970,5.335,148.919
C04514=1225.255,-46.038,-39.074,-179.973,5.335,148.919
C04515=1225.259,-46.289,-39.062,-179.975,5.335,148.920
C04516=1225.265,-46.538,-39.049,-179.977,5.335,148.921
C04517=1225.270,-46.787,-39.036,-179.980,5.334,148.921
C04518=1225.275,-47.037,-39.024,-179.982,5.335,148.922
C04519=1225.280,-47.287,-39.012,-179.985,5.334,148.923
C04520=1225.285,-47.537,-38.999,-179.987,5.334,148.923
C04521=1225.290,-47.786,-38.986,-179.990,5.334,148.924
C04522=1225.296,-48.036,-38.974,-179.992,5.333,148.925
C04523=1225.301,-48.306,-38.960,-179.995,5.334,148.926
C04524=1225.307,-48.575,-38.947,-179.997,5.334,148.927
C04525=1225.312,-48.845,-38.934,180.000,5.333,148.927
C04526=1225.318,-49.115,-38.920,179.997,5.333,148.928
C04527=1225.323,-49.365,-38.907,179.995,5.333,148.929
C04528=1225.328,-49.615,-38.895,179.992,5.333,148.929
C04529=1225.333,-49.864,-38.883,179.990,5.333,148.930
C04530=1225.339,-50.113,-38.870,179.988,5.332,148.931
C04531=1225.344,-50.363,-38.858,179.986,5.333,148.931
C04532=1225.349,-50.612,-38.845,179.983,5.332,148.932
C04533=1225.354,-50.863,-38.833,179.980,5.332,148.933
C04534=1225.359,-51.112,-38.821,179.978,5.332,148.934
C04535=1225.363,-51.361,-38.809,179.976,5.332,148.934
C04536=1225.369,-51.611,-38.797,179.973,5.332,148.935
C04537=1225.374,-51.861,-38.784,179.971,5.332,148.936
C04538=1225.379,-52.111,-38.772,179.968,5.331,148.936
C04539=1225.384,-52.360,-38.760,179.966,5.331,148.937
C04540=1225.389,-52.610,-38.747,179.963,5.331,148.938
C04541=1225.394,-52.860,-38.735,179.961,5.331,148.938
C04542=1225.400,-53.109,-38.722,179.959,5.331,148.939
C04543=1225.405,-53.359,-38.710,179.957,5.331,148.940
C04544=1225.410,-53.608,-38.698,179.954,5.331,148.941
C04545=1225.416,-53.858,-38.686,179.951,5.330,148.941
C04546=1225.421,-54.108,-38.673,179.949,5.330,148.942
C04547=1225.426,-54.358,-38.661,179.946,5.330,148.943
C04548=1225.430,-54.607,-38.649,179.944,5.330,148.943
C04549=1225.435,-54.857,-38.637,179.942,5.330,148.944
C04550=1225.440,-55.107,-38.624,179.939,5.329,148.945
C04551=1225.446,-55.357,-38.613,179.937,5.330,148.946
C04552=1225.451,-55.606,-38.600,179.934,5.329,148.946
C04553=1225.456,-55.856,-38.588,179.932,5.330,148.947
C04554=1225.462,-56.105,-38.575,179.930,5.329,148.948
C04555=1225.466,-56.355,-38.564,179.927,5.329,148.948
C04556=1225.471,-56.604,-38.552,179.925,5.329,148.949
C04557=1225.477,-56.854,-38.540,179.922,5.328,148.950
C04558=1225.482,-57.103,-38.527,179.920,5.329,148.950
C04559=1225.487,-57.353,-38.515,179.917,5.328,148.951
C04560=1225.492,-57.603,-38.503,179.915,5.329,148.952
C04561=1225.497,-57.852,-38.491,179.913,5.328,148.953
C04562=1225.503,-58.102,-38.479,179.910,5.329,148.953
C04563=1225.508,-58.351,-38.467,179.908,5.328,148.954
C04564=1225.513,-58.602,-38.455,179.905,5.328,148.955
C04565=1225.518,-58.851,-38.442,179.903,5.328,148.955
C04566=1225.522,-59.101,-38.431,179.900,5.327,148.956
C04567=1225.528,-59.351,-38.419,179.898,5.328,148.957
C04568=1225.533,-59.600,-38.406,179.896,5.327,148.958
C04569=1225.538,-59.850,-38.394,179.894,5.328,148.958
C04570=1225.543,-60.100,-38.382,179.891,5.327,148.959
C04571=1225.548,-60.349,-38.370,179.889,5.328,148.960
C04572=1225.554,-60.599,-38.359,179.886,5.327,148.960
C04573=1225.559,-60.848,-38.346,179.883,5.327,148.961
C04574=1225.564,-61.098,-38.334,179.881,5.327,148.962
C04575=1225.569,-61.348,-38.323,179.879,5.326,148.962
C04576=1225.574,-61.597,-38.310,179.877,5.327,148.963
C04577=1225.579,-61.847,-38.298,179.874,5.326,148.964
C04578=1225.585,-62.097,-38.286,179.872,5.327,148.965
C04579=1225.590,-62.347,-38.275,179.869,5.326,148.965
C04580=1225.595,-62.596,-38.263,179.867,5.327,148.966
C04581=1225.600,-62.846,-38.251,179.864,5.326,148.967
C04582=1225.605,-63.096,-38.239,179.862,5.326,148.967
C04583=1225.610,-63.345,-38.227,179.860,5.326,148.968
C04584=1225.615,-63.595,-38.215,179.857,5.325,148.969
C04585=1225.621,-63.845,-38.203,179.855,5.326,148.970
C04586=1225.625,-64.095,-38.192,179.852,5.325,148.970
C04587=1225.631,-64.343,-38.179,179.850,5.326,148.971
C04588=1225.637,-64.593,-38.168,179.848,5.325,148.972
C04589=1225.641,-64.843,-38.156,179.845,5.326,148.972
C04590=1225.647,-65.093,-38.144,179.843,5.325,148.973
C04591=1225.652,-65.343,-38.132,179.840,5.325,148.974
C04592=1225.657,-65.592,-38.120,179.838,5.325,148.974
C04593=1225.662,-65.842,-38.109,179.835,5.325,148.975
C04594=1225.667,-66.091,-38.097,179.833,5.325,148.976
C04595=1225.672,-66.341,-38.085,179.831,5.324,148.977
C04596=1225.678,-66.591,-38.074,179.828,5.325,148.977
C04597=1225.683,-66.840,-38.061,179.826,5.324,148.978
C04598=1225.687,-67.090,-38.050,179.824,5.325,148.979
C04599=1225.693,-67.340,-38.038,179.821,5.324,148.979
C04600=1225.698,-67.590,-38.026,179.819,5.324,148.980
C04601=1225.703,-67.839,-38.015,179.816,5.324,148.981
C04602=1225.709,-68.089,-38.003,179.814,5.324,148.982
C04603=1225.714,-68.338,-37.992,179.812,5.324,148.982
C04604=1225.719,-68.588,-37.980,179.809,5.323,148.983
C04605=1225.724,-68.838,-37.967,179.807,5.324,148.984
C04606=1225.729,-69.087,-37.956,179.804,5.323,148.984
C04607=1225.734,-69.337,-37.944,179.802,5.324,148.985
C04608=1225.739,-69.587,-37.933,179.799,5.323,148.986
C04609=1225.744,-69.837,-37.921,179.797,5.324,148.986
C04610=1225.750,-70.087,-37.909,179.795,5.323,148.987
C04611=1225.755,-70.336,-37.898,179.793,5.323,148.988
C04612=1225.761,-70.585,-37.886,179.790,5.323,148.989
C04613=1225.765,-70.835,-37.875,179.787,5.323,148.989
C04614=1225.771,-71.085,-37.863,179.785,5.323,148.990
C04615=1225.775,-71.335,-37.852,179.782,5.322,148.991
C04616=1225.781,-71.585,-37.840,179.780,5.323,148.991
C04617=1225.786,-71.835,-37.828,179.778,5.322,148.992
C04618=1225.792,-72.083,-37.817,179.776,5.323,148.993
C04619=1225.797,-72.333,-37.805,179.773,5.322,148.993
C04620=1225.802,-72.583,-37.794,179.771,5.322,148.994
C04621=1225.807,-72.833,-37.782,179.769,5.322,148.995
C04622=1225.812,-73.083,-37.771,179.767,5.322,148.995
C04623=1225.817,-73.333,-37.759,179.764,5.322,148.996
C04624=1225.822,-73.581,-37.748,179.762,5.322,148.997
C04625=1225.828,-73.831,-37.736,179.759,5.321,148.998
C04626=1225.833,-74.081,-37.725,179.757,5.322,148.998
C04627=1225.838,-74.351,-37.712,179.754,5.322,148.999
C04628=1225.844,-74.622,-37.700,179.751,5.321,149.000
C04629=1225.849,-74.892,-37.687,179.749,5.322,149.001
C04630=1225.855,-75.163,-37.675,179.746,5.321,149.001
C04631=1225.860,-75.412,-37.664,179.744,5.321,149.002
C04632=1225.866,-75.662,-37.652,179.742,5.321,149.003
C04633=1225.870,-75.911,-37.641,179.739,5.321,149.003
C04634=1225.876,-76.161,-37.629,179.737,5.321,149.004
C04635=1225.881,-76.411,-37.617,179.734,5.320,149.005
C04636=1225.887,-76.660,-37.606,179.732,5.321,149.006
C04637=1225.891,-76.910,-37.595,179.729,5.320,149.006
C04638=1225.897,-77.160,-37.583,179.727,5.321,149.007
C04639=1225.902,-77.410,-37.572,179.725,5.320,149.008
C04640=1225.907,-77.659,-37.561,179.723,5.321,149.008
C04641=1225.912,-77.909,-37.549,179.720,5.320,149.009
C04642=1225.917,-78.159,-37.538,179.718,5.321,149.010
C04643=1225.923,-78.409,-37.526,179.715,5.320,149.011
C04644=1225.927,-78.658,-37.515,179.713,5.320,149.011
C04645=1225.934,-78.908,-37.504,179.710,5.320,149.012
C04646=1225.938,-79.158,-37.493,179.708,5.320,149.013
C04647=1225.943,-79.407,-37.481,179.706,5.320,149.013
C04648=1225.948,-79.657,-37.470,179.704,5.320,149.014
C04649=1225.954,-79.906,-37.459,179.701,5.320,149.015
C04650=1225.959,-80.156,-37.448,179.699,5.319,149.015
C04651=1225.964,-80.406,-37.436,179.697,5.319,149.016
C04652=1225.969,-80.656,-37.425,179.694,5.319,149.017
C04653=1225.975,-80.905,-37.413,179.692,5.319,149.017
C04654=1225.980,-81.155,-37.403,179.689,5.319,149.018
C04655=1225.985,-81.405,-37.392,179.687,5.319,149.019
C04656=1225.991,-81.654,-37.380,179.684,5.319,149.020
C04657=1225.995,-81.904,-37.369,179.682,5.319,149.020
C04658=1226.000,-82.154,-37.358,179.680,5.319,149.021
C04659=1226.006,-82.404,-37.346,179.678,5.319,149.022
C04660=1226.011,-82.653,-37.335,179.675,5.318,149.022
C04661=1226.016,-82.903,-37.324,179.673,5.319,149.023
C04662=1226.021,-83.153,-37.313,179.670,5.318,149.024
C04663=1226.026,-83.403,-37.302,179.668,5.319,149.025
C04664=1226.031,-83.652,-37.291,179.665,5.318,149.025
C04665=1226.036,-83.902,-37.280,179.663,5.319,149.026
C04666=1226.042,-84.152,-37.268,179.661,5.318,149.027
C04667=1226.047,-84.401,-37.257,179.659,5.318,149.027
C04668=1226.052,-84.651,-37.247,179.656,5.318,149.028
C04669=1226.057,-84.901,-37.235,179.654,5.318,149.029
C04670=1226.063,-85.150,-37.224,179.651,5.318,149.029
C04671=1226.068,-85.400,-37.213,179.649,5.318,149.030
C04672=1226.073,-85.650,-37.202,179.646,5.318,149.031
C04673=1226.079,-85.899,-37.191,179.645,5.318,149.031
C04674=1226.084,-86.149,-37.180,179.642,5.317,149.032
C04675=1226.088,-86.399,-37.169,179.640,5.318,149.033
C04676=1226.094,-86.648,-37.158,179.637,5.317,149.034
C04677=1226.099,-86.898,-37.147,179.635,5.318,149.034
C04678=1226.104,-87.148,-37.135,179.633,5.317,149.035
C04679=1226.110,-87.398,-37.125,179.630,5.318,149.036
C04680=1226.114,-87.647,-37.114,179.628,5.317,149.036
C04681=1226.119,-87.897,-37.102,179.626,5.317,149.037
C04682=1226.125,-88.147,-37.092,179.623,5.317,149.038
C04683=1226.130,-88.396,-37.080,179.621,5.317,149.039
C04684=1226.135,-88.647,-37.070,179.618,5.317,149.039
C04685=1226.140,-88.895,-37.059,179.616,5.317,149.040
C04686=1226.145,-89.146,-37.048,179.613,5.317,149.041
C04687=1226.151,-89.395,-37.037,179.611,5.317,149.041
C04688=1226.156,-89.645,-37.026,179.609,5.317,149.042
C04689=1226.161,-89.895,-37.015,179.607,5.317,149.043
C04690=1226.167,-90.144,-37.005,179.604,5.317,149.043
C04691=1226.171,-90.394,-36.993,179.602,5.317,149.044
C04692=1226.177,-90.644,-36.983,179.600,5.316,149.045
C04693=1226.182,-90.893,-36.971,179.598,5.317,149.045
C04694=1226.187,-91.144,-36.961,179.595,5.316,149.046
C04695=1226.193,-91.393,-36.950,179.593,5.316,149.047
C04696=1226.198,-91.643,-36.939,179.590,5.316,149.048
C04697=1226.203,-91.892,-36.928,179.588,5.316,149.048
C04698=1226.208,-92.142,-36.918,179.585,5.316,149.049
C04699=1226.213,-92.392,-36.906,179.583,5.316,149.050
C04700=1226.219,-92.642,-36.896,179.581,5.316,149.050
C04701=1226.224,-92.891,-36.884,179.579,5.316,149.051
C04702=1226.229,-93.141,-36.874,179.576,5.316,149.052
C04703=1226.234,-93.390,-36.863,179.574,5.316,149.053
C04704=1226.239,-93.640,-36.853,179.571,5.316,149.053
C04705=1226.244,-93.890,-36.842,179.569,5.316,149.054
C04706=1226.249,-94.140,-36.831,179.567,5.315,149.054
C04707=1226.255,-94.389,-36.821,179.565,5.316,149.055
C04708=1226.259,-94.639,-36.809,179.562,5.315,149.056
C04709=1226.266,-94.889,-36.799,179.560,5.315,149.057
C04710=1226.271,-95.139,-36.788,179.557,5.315,149.057
C04711=1226.276,-95.388,-36.777,179.555,5.315,149.058
C04712=1226.281,-95.638,-36.766,179.553,5.315,149.059
C04713=1226.287,-95.888,-36.756,179.550,5.315,149.059
C04714=1226.291,-96.137,-36.745,179.548,5.315,149.060
C04715=1226.297,-96.387,-36.735,179.546,5.315,149.061
C04716=1226.302,-96.637,-36.724,179.543,5.315,149.062
C04717=1226.307,-96.887,-36.713,179.541,5.315,149.062
C04718=1226.312,-97.136,-36.703,179.538,5.315,149.063
C04719=1226.317,-97.387,-36.692,179.537,5.315,149.063
C04720=1226.323,-97.635,-36.681,179.534,5.314,149.064
C04721=1226.328,-97.886,-36.671,179.532,5.315,149.065
C04722=1226.333,-98.135,-36.660,179.529,5.314,149.066
C04723=1226.338,-98.385,-36.649,179.527,5.315,149.066
C04724=1226.343,-98.634,-36.639,179.525,5.315,149.067
C04725=1226.348,-98.885,-36.628,179.522,5.314,149.068
C04726=1226.354,-99.134,-36.618,179.520,5.315,149.068
C04727=1226.359,-99.384,-36.607,179.518,5.314,149.069
C04728=1226.364,-99.633,-36.597,179.515,5.315,149.070
C04729=1226.369,-99.884,-36.586,179.513,5.314,149.071
C04730=1226.375,-100.133,-36.576,179.511,5.315,149.071
C04731=1226.381,-100.404,-36.564,179.508,5.314,149.072
C04732=1226.386,-100.675,-36.553,179.505,5.314,149.073
C04733=1226.392,-100.946,-36.541,179.503,5.314,149.073
C04734=1226.397,-101.217,-36.530,179.501,5.314,149.074
C04735=1226.403,-101.467,-36.520,179.498,5.314,149.075
C04736=1226.408,-101.717,-36.509,179.496,5.314,149.076
C04737=1226.413,-101.966,-36.498,179.494,5.314,149.076
C04738=1226.418,-102.216,-36.488,179.491,5.314,149.077
C04739=1226.424,-102.466,-36.477,179.489,5.314,149.078
C04740=1226.429,-102.716,-36.467,179.486,5.314,149.078
C04741=1226.434,-102.965,-36.457,179.484,5.314,149.079
C04742=1226.440,-103.215,-36.446,179.482,5.313,149.080
C04743=1226.444,-103.464,-36.435,179.480,5.313,149.080
C04744=1226.450,-103.714,-36.425,179.477,5.313,149.081
C04745=1226.454,-103.964,-36.415,179.475,5.313,149.082
C04746=1226.460,-104.213,-36.405,179.472,5.313,149.082
C04747=1226.465,-104.464,-36.394,179.470,5.313,149.083
C04748=1226.471,-104.713,-36.384,179.468,5.314,149.084
C04749=1226.476,-104.963,-36.374,179.466,5.313,149.085
C04750=1226.481,-105.212,-36.362,179.463,5.314,149.085
C04751=1226.486,-105.462,-36.352,179.461,5.313,149.086
C04752=1226.491,-105.712,-36.342,179.459,5.313,149.087
C04753=1226.496,-105.961,-36.332,179.457,5.313,149.087
C04754=1226.502,-106.211,-36.322,179.454,5.313,149.088
C04755=1226.507,-106.461,-36.311,179.452,5.313,149.089
C04756=1226.512,-106.711,-36.301,179.450,5.313,149.089
C04757=1226.517,-106.961,-36.290,179.447,5.313,149.090
C04758=1226.523,-107.211,-36.280,179.445,5.313,149.091
C04759=1226.529,-107.460,-36.270,179.442,5.313,149.092
C04760=1226.533,-107.710,-36.260,179.440,5.313,149.092
C04761=1226.539,-107.960,-36.250,179.438,5.312,149.093
C04762=1226.544,-108.210,-36.239,179.436,5.312,149.093
C04763=1226.549,-108.459,-36.229,179.433,5.312,149.094
C04764=1226.555,-108.709,-36.219,179.431,5.312,149.095
C04765=1226.559,-108.959,-36.209,179.429,5.313,149.096
C04766=1226.565,-109.208,-36.199,179.426,5.312,149.096
C04767=1226.570,-109.458,-36.188,179.424,5.313,149.097
C04768=1226.575,-109.708,-36.178,179.422,5.312,149.098
C04769=1226.581,-109.958,-36.168,179.419,5.313,149.098
C04770=1226.586,-110.207,-36.158,179.417,5.312,149.099
C04771=1226.591,-110.457,-36.147,179.415,5.312,149.100
C04772=1226.596,-110.707,-36.137,179.412,5.312,149.100
C04773=1226.602,-110.956,-36.127,179.410,5.312,149.101
C04774=1226.607,-111.207,-36.116,179.408,5.312,149.102
C04775=1226.612,-111.456,-36.107,179.406,5.312,149.103
C04776=1226.617,-111.705,-36.097,179.403,5.312,149.103
C04777=1226.622,-111.956,-36.086,179.401,5.312,149.104
C04778=1226.628,-112.205,-36.076,179.399,5.312,149.104
C04779=1226.633,-112.454,-36.066,179.397,5.312,149.105
C04780=1226.638,-112.705,-36.056,179.394,5.312,149.106
C04781=1226.644,-112.955,-36.046,179.392,5.312,149.107
C04782=1226.649,-113.204,-36.037,179.390,5.312,149.107
C04783=1226.654,-113.454,-36.026,179.387,5.312,149.108
C04784=1226.659,-113.704,-36.016,179.385,5.312,149.109
C04785=1226.665,-113.953,-36.006,179.382,5.311,149.109
C04786=1226.669,-114.203,-35.996,179.381,5.311,149.110
C04787=1226.675,-114.453,-35.985,179.378,5.311,149.111
C04788=1226.680,-114.702,-35.975,179.376,5.311,149.111
C04789=1226.685,-114.952,-35.966,179.373,5.311,149.112
C04790=1226.690,-115.202,-35.956,179.371,5.311,149.113
C04791=1226.696,-115.452,-35.945,179.369,5.312,149.113
C04792=1226.701,-115.701,-35.936,179.366,5.311,149.114
C04793=1226.706,-115.951,-35.926,179.365,5.311,149.115
C04794=1226.711,-116.201,-35.915,179.362,5.311,149.115
C04795=1226.717,-116.451,-35.906,179.360,5.311,149.116
C04796=1226.722,-116.700,-35.896,179.357,5.311,149.117
C04797=1226.727,-116.951,-35.885,179.355,5.311,149.118
C04798=1226.732,-117.200,-35.876,179.353,5.311,149.118
C04799=1226.738,-117.450,-35.866,179.350,5.311,149.119
C04800=1226.744,-117.700,-35.856,179.348,5.310,149.119
C04801=1226.748,-117.950,-35.846,179.346,5.311,149.120
C04802=1226.753,-118.199,-35.836,179.344,5.311,149.121
C04803=1226.759,-118.449,-35.826,179.341,5.311,149.122
C04804=1226.764,-118.698,-35.817,179.339,5.311,149.122
C04805=1226.769,-118.949,-35.806,179.337,5.311,149.123
C04806=1226.774,-119.198,-35.797,179.335,5.311,149.124
C04807=1226.780,-119.448,-35.787,179.332,5.310,149.124
C04808=1226.786,-119.698,-35.777,179.330,5.311,149.125
C04809=1226.790,-119.947,-35.767,179.328,5.310,149.126
C04810=1226.795,-120.197,-35.757,179.325,5.311,149.126
C04811=1226.801,-120.447,-35.748,179.323,5.310,149.127
C04812=1226.806,-120.696,-35.738,179.321,5.310,149.128
C04813=1226.812,-120.946,-35.727,179.319,5.310,149.128
C04814=1226.816,-121.197,-35.718,179.316,5.310,149.129
C04815=1226.822,-121.446,-35.708,179.314,5.310,149.130
C04816=1226.827,-121.695,-35.698,179.312,5.310,149.130
C04817=1226.833,-121.946,-35.689,179.310,5.310,149.131
C04818=1226.838,-122.195,-35.679,179.307,5.310,149.132
C04819=1226.843,-122.445,-35.669,179.305,5.310,149.133
C04820=1226.848,-122.695,-35.660,179.303,5.310,149.133
C04821=1226.853,-122.944,-35.649,179.300,5.310,149.134
C04822=1226.858,-123.194,-35.640,179.298,5.310,149.135
C04823=1226.864,-123.444,-35.630,179.296,5.310,149.135
C04824=1226.869,-123.693,-35.621,179.294,5.310,149.136
C04825=1226.874,-123.944,-35.611,179.291,5.310,149.137
C04826=1226.880,-124.193,-35.601,179.289,5.310,149.137
C04827=1226.885,-124.443,-35.591,179.287,5.309,149.138
C04828=1226.891,-124.693,-35.582,179.285,5.310,149.139
C04829=1226.895,-124.942,-35.572,179.282,5.309,149.139
C04830=1226.901,-125.192,-35.562,179.280,5.310,149.140
C04831=1226.906,-125.442,-35.553,179.278,5.309,149.141
C04832=1226.911,-125.692,-35.543,179.275,5.309,149.141
C04833=1226.916,-125.942,-35.533,179.273,5.310,149.142
C04834=1226.921,-126.191,-35.524,179.271,5.309,149.143
C04835=1226.500,-126.202,-35.560,179.266,5.313,149.145
C04836=1226.495,-125.952,-35.570,179.269,5.313,149.144
C04837=1226.489,-125.702,-35.579,179.271,5.313,149.143
C04838=1226.484,-125.453,-35.589,179.273,5.313,149.143
C04839=1226.479,-125.202,-35.598,179.276,5.313,149.142
C04840=1226.474,-124.953,-35.608,179.278,5.313,149.141
C04841=1226.469,-124.704,-35.618,179.280,5.313,149.141
C04842=1226.463,-124.453,-35.627,179.282,5.313,149.140
C04843=1226.458,-124.204,-35.637,179.285,5.313,149.139
C04844=1226.452,-123.954,-35.647,179.287,5.313,149.139
C04845=1226.448,-123.704,-35.657,179.290,5.313,149.138
C04846=1226.442,-123.455,-35.667,179.292,5.313,149.137
C04847=1226.437,-123.205,-35.676,179.293,5.313,149.137
C04848=1226.432,-122.955,-35.686,179.296,5.313,149.136
C04849=1226.426,-122.705,-35.695,179.298,5.313,149.135
C04850=1226.421,-122.456,-35.705,179.301,5.314,149.134
C04851=1226.416,-122.206,-35.715,179.303,5.313,149.134
C04852=1226.411,-121.956,-35.724,179.306,5.314,149.133
C04853=1226.406,-121.706,-35.734,179.307,5.314,149.133
C04854=1226.400,-121.457,-35.744,179.310,5.314,149.132
C04855=1226.394,-121.207,-35.754,179.312,5.314,149.131
C04856=1226.390,-120.957,-35.764,179.315,5.314,149.130
C04857=1226.384,-120.707,-35.774,179.317,5.314,149.130
C04858=1226.379,-120.457,-35.783,179.319,5.313,149.129
C04859=1226.374,-120.208,-35.793,179.321,5.314,149.129
C04860=1226.369,-119.959,-35.803,179.323,5.314,149.128
C04861=1226.363,-119.708,-35.813,179.326,5.314,149.127
C04862=1226.358,-119.458,-35.823,179.328,5.314,149.126
C04863=1226.353,-119.209,-35.832,179.331,5.314,149.126
C04864=1226.347,-118.959,-35.843,179.333,5.314,149.125
C04865=1226.343,-118.709,-35.852,179.335,5.315,149.124
C04866=1226.337,-118.459,-35.862,179.337,5.314,149.124
C04867=1226.332,-118.210,-35.872,179.339,5.314,149.123
C04868=1226.327,-117.961,-35.882,179.342,5.314,149.122
C04869=1226.321,-117.710,-35.892,179.344,5.314,149.122
C04870=1226.317,-117.460,-35.901,179.346,5.314,149.121
C04871=1226.311,-117.211,-35.912,179.349,5.314,149.120
C04872=1226.305,-116.961,-35.922,179.351,5.315,149.120
C04873=1226.301,-116.711,-35.931,179.353,5.314,149.119
C04874=1226.295,-116.461,-35.941,179.356,5.315,149.118
C04875=1226.290,-116.212,-35.951,179.358,5.314,149.118
C04876=1226.285,-115.963,-35.961,179.360,5.315,149.117
C04877=1226.280,-115.712,-35.972,179.362,5.314,149.116
C04878=1226.274,-115.462,-35.981,179.365,5.315,149.115
C04879=1226.269,-115.213,-35.991,179.367,5.315,149.115
C04880=1226.263,-114.963,-36.001,179.369,5.315,149.114
C04881=1226.258,-114.713,-36.011,179.371,5.315,149.113
C04882=1226.254,-114.464,-36.021,179.374,5.315,149.113
C04883=1226.248,-114.214,-36.031,179.376,5.315,149.112
C04884=1226.243,-113.963,-36.041,179.378,5.315,149.111
C04885=1226.237,-113.714,-36.051,179.381,5.315,149.111
C04886=1226.232,-113.465,-36.061,179.383,5.315,149.110
C04887=1226.227,-113.215,-36.071,179.385,5.315,149.109
C04888=1226.222,-112.965,-36.082,179.387,5.315,149.109
C04889=1226.217,-112.716,-36.091,179.390,5.316,149.108
C04890=1226.211,-112.466,-36.102,179.392,5.315,149.107
C04891=1226.206,-112.216,-36.112,179.394,5.315,149.107
C04892=1226.201,-111.966,-36.122,179.397,5.315,149.106
C04893=1226.195,-111.716,-36.131,179.399,5.315,149.105
C04894=1226.190,-111.466,-36.142,179.401,5.316,149.105
C04895=1226.185,-111.217,-36.152,179.403,5.315,149.104
C04896=1226.179,-110.967,-36.162,179.406,5.316,149.103
C04897=1226.175,-110.717,-36.172,179.408,5.315,149.102
C04898=1226.169,-110.468,-36.182,179.411,5.316,149.102
C04899=1226.164,-110.218,-36.193,179.413,5.315,149.101
C04900=1226.159,-109.968,-36.203,179.415,5.316,149.100
C04901=1226.153,-109.718,-36.213,179.418,5.315,149.100
C04902=1226.148,-109.469,-36.223,179.420,5.316,149.099
C04903=1226.143,-109.219,-36.234,179.422,5.316,149.098
C04904=1226.138,-108.969,-36.244,179.425,5.316,149.098
C04905=1226.132,-108.720,-36.254,179.427,5.316,149.097
C04906=1226.127,-108.470,-36.265,179.429,5.316,149.096
C04907=1226.122,-108.220,-36.274,179.431,5.316,149.096
C04908=1226.117,-107.970,-36.285,179.433,5.316,149.095
C04909=1226.112,-107.720,-36.295,179.436,5.316,149.094
C04910=1226.106,-107.471,-36.305,179.438,5.316,149.094
C04911=1226.101,-107.221,-36.316,179.440,5.317,149.093
C04912=1226.096,-106.971,-36.325,179.443,5.316,149.092
C04913=1226.091,-106.722,-36.336,179.445,5.317,149.091
C04914=1226.086,-106.472,-36.346,179.447,5.316,149.091
C04915=1226.080,-106.222,-36.356,179.450,5.317,149.090
C04916=1226.075,-105.972,-36.367,179.452,5.316,149.089
C04917=1226.070,-105.723,-36.378,179.455,5.317,149.089
C04918=1226.064,-105.473,-36.388,179.457,5.316,149.088
C04919=1226.060,-105.223,-36.398,179.460,5.317,149.087
C04920=1226.054,-104.974,-36.408,179.461,5.317,149.087
C04921=1226.049,-104.724,-36.419,179.464,5.317,149.086
C04922=1226.044,-104.474,-36.429,179.466,5.317,149.085
C04923=1226.039,-104.224,-36.440,179.468,5.316,149.085
C04924=1226.033,-103.974,-36.450,179.471,5.317,149.084
C04925=1226.027,-103.725,-36.460,179.473,5.317,149.083
C04926=1226.023,-103.475,-36.471,179.475,5.317,149.082
C04927=1226.017,-103.226,-36.482,179.478,5.317,149.082
C04928=1226.013,-102.976,-36.492,179.480,5.317,149.081
C04929=1226.007,-102.726,-36.502,179.482,5.317,149.081
C04930=1226.002,-102.476,-36.512,179.484,5.317,149.080
C04931=1225.997,-102.226,-36.523,179.487,5.317,149.079
C04932=1225.991,-101.977,-36.533,179.489,5.318,149.078
C04933=1225.986,-101.727,-36.544,179.491,5.317,149.078
C04934=1225.981,-101.478,-36.554,179.494,5.318,149.077
C04935=1225.976,-101.227,-36.565,179.496,5.317,149.076
C04936=1225.971,-100.956,-36.576,179.499,5.318,149.076
C04937=1225.964,-100.686,-36.588,179.501,5.317,149.075
C04938=1225.958,-100.414,-36.599,179.504,5.318,149.074
C04939=1225.954,-100.144,-36.611,179.507,5.318,149.073
C04940=1225.948,-99.894,-36.621,179.508,5.318,149.073
C04941=1225.943,-99.644,-36.632,179.511,5.318,149.072
C04942=1225.937,-99.394,-36.642,179.513,5.318,149.071
C04943=1225.933,-99.145,-36.653,179.516,5.318,149.071
C04944=1225.927,-98.895,-36.663,179.518,5.318,149.070
C04945=1225.922,-98.645,-36.674,179.521,5.318,149.069
C04946=1225.917,-98.395,-36.684,179.523,5.318,149.068
C04947=1225.912,-98.146,-36.695,179.525,5.318,149.068
C04948=1225.906,-97.896,-36.706,179.527,5.318,149.067
C04949=1225.901,-97.646,-36.716,179.529,5.318,149.066
C04950=1225.896,-97.397,-36.727,179.532,5.318,149.066
C04951=1225.891,-97.147,-36.738,179.534,5.318,149.065
C04952=1225.885,-96.897,-36.748,179.536,5.319,149.064
C04953=1225.881,-96.648,-36.759,179.539,5.318,149.064
C04954=1225.875,-96.398,-36.769,179.541,5.319,149.063
C04955=1225.870,-96.148,-36.780,179.543,5.318,149.062
C04956=1225.865,-95.899,-36.791,179.546,5.319,149.062
C04957=1225.860,-95.649,-36.801,179.548,5.318,149.061
C04958=1225.854,-95.399,-36.812,179.551,5.319,149.060
C04959=1225.849,-95.149,-36.824,179.553,5.319,149.059
C04960=1225.843,-94.900,-36.834,179.555,5.319,149.059
C04961=1225.838,-94.649,-36.844,179.558,5.319,149.058
C04962=1225.833,-94.400,-36.855,179.560,5.319,149.057
C04963=1225.828,-94.150,-36.866,179.562,5.319,149.057
C04964=1225.823,-93.901,-36.877,179.565,5.320,149.056
C04965=1225.818,-93.651,-36.887,179.567,5.319,149.055
C04966=1225.813,-93.401,-36.898,179.569,5.320,149.055
C04967=1225.807,-93.152,-36.909,179.571,5.319,149.054
C04968=1225.802,-92.902,-36.919,179.574,5.320,149.053
C04969=1225.797,-92.653,-36.930,179.576,5.319,149.052
C04970=1225.791,-92.402,-36.942,179.579,5.320,149.052
C04971=1225.786,-92.153,-36.952,179.581,5.319,149.051
C04972=1225.781,-91.903,-36.963,179.584,5.320,149.050
C04973=1225.776,-91.653,-36.974,179.586,5.319,149.050
C04974=1225.771,-91.404,-36.985,179.588,5.320,149.049
C04975=1225.766,-91.154,-36.995,179.590,5.320,149.048
C04976=1225.760,-90.905,-37.006,179.593,5.320,149.047
C04977=1225.755,-90.654,-37.017,179.595,5.320,149.047
C04978=1225.750,-90.404,-37.028,179.598,5.320,149.046
C04979=1225.744,-90.155,-37.039,179.599,5.320,149.046
C04980=1225.740,-89.905,-37.050,179.602,5.321,149.045
C04981=1225.734,-89.656,-37.060,179.604,5.320,149.044
C04982=1225.729,-89.406,-37.071,179.607,5.321,149.043
C04983=1225.724,-89.156,-37.083,179.609,5.320,149.043
C04984=1225.718,-88.907,-37.094,179.612,5.321,149.042
C04985=1225.713,-88.656,-37.104,179.614,5.320,149.041
C04986=1225.709,-88.407,-37.115,179.616,5.321,149.041
C04987=1225.703,-88.158,-37.126,179.619,5.320,149.040
C04988=1225.698,-87.907,-37.138,179.621,5.321,149.039
C04989=1225.692,-87.658,-37.148,179.623,5.321,149.038
C04990=1225.687,-87.408,-37.159,179.626,5.321,149.038
C04991=1225.683,-87.158,-37.170,179.628,5.321,149.037
C04992=1225.677,-86.909,-37.181,179.631,5.321,149.036
C04993=1225.672,-86.659,-37.192,179.633,5.321,149.036
C04994=1225.667,-86.409,-37.204,179.636,5.321,149.035
C04995=1225.661,-86.160,-37.214,179.637,5.321,149.034
C04996=1225.657,-85.910,-37.225,179.640,5.322,149.034
C04997=1225.651,-85.660,-37.237,179.642,5.321,149.033
C04998=1225.646,-85.411,-37.247,179.645,5.322,149.032
C04999=1225.641,-85.161,-37.259,179.647,5.321,149.032
C05000=1225.636,-84.911,-37.269,179.649,5.322,149.031
C05001=1225.630,-84.662,-37.281,179.651,5.321,149.030
C05002=1225.625,-84.412,-37.292,179.654,5.322,149.029
C05003=1225.620,-84.162,-37.303,179.656,5.322,149.029
C05004=1225.614,-83.912,-37.314,179.659,5.322,149.028
C05005=1225.609,-83.663,-37.325,179.661,5.322,149.027
C05006=1225.605,-83.413,-37.337,179.664,5.322,149.027
C05007=1225.600,-83.163,-37.347,179.666,5.322,149.026
C05008=1225.594,-82.914,-37.359,179.668,5.322,149.025
C05009=1225.589,-82.664,-37.370,179.670,5.322,149.025
C05010=1225.584,-82.414,-37.381,179.673,5.322,149.024
C05011=1225.578,-82.165,-37.392,179.675,5.322,149.023
C05012=1225.573,-81.915,-37.403,179.678,5.322,149.022
C05013=1225.569,-81.665,-37.415,179.680,5.322,149.022
C05014=1225.563,-81.415,-37.426,179.683,5.323,149.021
C05015=1225.558,-81.166,-37.437,179.685,5.322,149.020
C05016=1225.553,-80.916,-37.448,179.687,5.323,149.020
C05017=1225.547,-80.666,-37.460,179.689,5.323,149.019
C05018=1225.542,-80.416,-37.471,179.692,5.323,149.018
C05019=1225.537,-80.167,-37.481,179.694,5.324,149.018
C05020=1225.532,-79.917,-37.493,179.696,5.323,149.017
C05021=1225.527,-79.668,-37.505,179.699,5.324,149.016
C05022=1225.521,-79.418,-37.515,179.701,5.323,149.016
C05023=1225.516,-79.168,-37.527,179.704,5.324,149.015
C05024=1225.511,-78.919,-37.538,179.706,5.323,149.014
C05025=1225.506,-78.669,-37.550,179.709,5.324,149.013
C05026=1225.501,-78.419,-37.561,179.711,5.324,149.013
C05027=1225.495,-78.170,-37.573,179.713,5.324,149.012
C05028=1225.490,-77.919,-37.583,179.715,5.324,149.011
C05029=1225.486,-77.670,-37.595,179.718,5.324,149.011
C05030=1225.480,-77.420,-37.606,179.720,5.324,149.010
C05031=1225.475,-77.171,-37.617,179.723,5.324,149.009
C05032=1225.469,-76.921,-37.629,179.725,5.324,149.008
C05033=1225.465,-76.671,-37.641,179.728,5.324,149.008
C05034=1225.459,-76.421,-37.652,179.730,5.324,149.007
C05035=1225.454,-76.173,-37.663,179.732,5.324,149.006
C05036=1225.449,-75.922,-37.674,179.735,5.324,149.006
C05037=1225.444,-75.672,-37.686,179.737,5.325,149.005
C05038=1225.439,-75.423,-37.697,179.739,5.324,149.004
C05039=1225.433,-75.173,-37.709,179.742,5.325,149.003
C05040=1225.428,-74.903,-37.722,179.745,5.325,149.003
C05041=1225.422,-74.632,-37.734,179.747,5.325,149.002
C05042=1225.417,-74.362,-37.747,179.749,5.325,149.001
C05043=1225.411,-74.092,-37.758,179.752,5.326,149.001
C05044=1225.406,-73.842,-37.770,179.754,5.325,149.000
C05045=1225.401,-73.592,-37.781,179.757,5.326,148.999
C05046=1225.396,-73.342,-37.793,179.759,5.325,148.998
C05047=1225.390,-73.093,-37.805,179.762,5.326,148.998
C05048=1225.385,-72.844,-37.816,179.764,5.326,148.997
C05049=1225.379,-72.594,-37.828,179.766,5.326,148.996
C05050=1225.375,-72.344,-37.839,179.768,5.326,148.996
C05051=1225.369,-72.094,-37.851,179.771,5.326,148.995
C05052=1225.365,-71.844,-37.862,179.773,5.326,148.994
C05053=1225.359,-71.594,-37.874,179.776,5.326,148.994
C05054=1225.354,-71.346,-37.885,179.778,5.326,148.993
C05055=1225.348,-71.096,-37.897,179.781,5.326,148.992
C05056=1225.344,-70.846,-37.908,179.783,5.327,148.991
C05057=1225.338,-70.596,-37.920,179.785,5.326,148.991
C05058=1225.334,-70.346,-37.932,179.788,5.327,148.990
C05059=1225.328,-70.096,-37.943,179.790,5.327,148.989
C05060=1225.323,-69.847,-37.955,179.793,5.327,148.989
C05061=1225.317,-69.598,-37.966,179.795,5.327,148.988
C05062=1225.312,-69.348,-37.978,179.798,5.327,148.987
C05063=1225.307,-69.098,-37.989,179.800,5.327,148.986
C05064=1225.302,-68.849,-38.002,179.802,5.327,148.986
C05065=1225.297,-68.599,-38.014,179.804,5.327,148.985
C05066=1225.292,-68.349,-38.025,179.807,5.327,148.984
C05067=1225.287,-68.099,-38.037,179.810,5.328,148.984
C05068=1225.282,-67.850,-38.048,179.812,5.327,148.983
C05069=1225.277,-67.600,-38.060,179.815,5.328,148.982
C05070=1225.271,-67.350,-38.072,179.817,5.328,148.982
C05071=1225.266,-67.101,-38.083,179.819,5.328,148.981
C05072=1225.261,-66.851,-38.096,179.821,5.328,148.980
C05073=1225.255,-66.602,-38.108,179.824,5.328,148.979
C05074=1225.251,-66.352,-38.119,179.826,5.328,148.979
C05075=1225.245,-66.102,-38.131,179.829,5.328,148.978
C05076=1225.240,-65.852,-38.143,179.831,5.328,148.977
C05077=1225.235,-65.602,-38.154,179.834,5.328,148.977
C05078=1225.230,-65.353,-38.166,179.836,5.329,148.976
C05079=1225.224,-65.103,-38.178,179.838,5.329,148.975
C05080=1225.220,-64.854,-38.190,179.841,5.329,148.974
C05081=1225.214,-64.604,-38.202,179.843,5.329,148.974
C05082=1225.209,-64.354,-38.214,179.846,5.329,148.973
C05083=1225.205,-64.105,-38.225,179.848,5.329,148.972
C05084=1225.199,-63.855,-38.237,179.850,5.329,148.972
C05085=1225.194,-63.605,-38.249,179.852,5.329,148.971
C05086=1225.189,-63.355,-38.260,179.855,5.330,148.970
C05087=1225.183,-63.107,-38.273,179.857,5.330,148.970
C05088=1225.178,-62.857,-38.285,179.859,5.330,148.969
C05089=1225.173,-62.607,-38.296,179.862,5.330,148.968
C05090=1225.168,-62.358,-38.308,179.864,5.330,148.968
C05091=1225.163,-62.108,-38.320,179.867,5.330,148.967
C05092=1225.157,-61.858,-38.332,179.869,5.330,148.966
C05093=1225.152,-61.608,-38.344,179.872,5.331,148.966
C05094=1225.147,-61.359,-38.356,179.874,5.330,148.965
C05095=1225.142,-61.109,-38.368,179.876,5.331,148.964
C05096=1225.136,-60.859,-38.380,179.879,5.331,148.963
C05097=1225.132,-60.610,-38.392,179.881,5.331,148.963
C05098=1225.127,-60.360,-38.404,179.884,5.331,148.962
C05099=1225.121,-60.110,-38.416,179.886,5.331,148.961
C05100=1225.116,-59.861,-38.428,179.889,5.331,148.961
C05101=1225.111,-59.611,-38.440,179.891,5.331,148.960
C05102=1225.106,-59.361,-38.451,179.893,5.332,148.959
C05103=1225.101,-59.112,-38.464,179.896,5.332,148.958
C05104=1225.096,-58.861,-38.476,179.898,5.332,148.958
C05105=1225.091,-58.612,-38.489,179.901,5.332,148.957
C05106=1225.086,-58.362,-38.500,179.903,5.332,148.956
C05107=1225.081,-58.112,-38.512,179.906,5.332,148.956
C05108=1225.076,-57.863,-38.525,179.908,5.332,148.955
C05109=1225.070,-57.613,-38.537,179.910,5.332,148.954
C05110=1225.065,-57.364,-38.549,179.912,5.332,148.954
C05111=1225.060,-57.114,-38.560,179.915,5.333,148.953
C05112=1225.055,-56.865,-38.573,179.918,5.333,148.952
C05113=1225.050,-56.615,-38.585,179.920,5.333,148.951
C05114=1225.044,-56.365,-38.597,179.922,5.333,148.951
C05115=1225.039,-56.116,-38.609,179.925,5.333,148.950
C05116=1225.034,-55.866,-38.621,179.927,5.333,148.949
C05117=1225.029,-55.616,-38.634,179.930,5.334,148.949
C05118=1225.024,-55.367,-38.645,179.932,5.334,148.948
C05119=1225.019,-55.117,-38.658,179.935,5.334,148.947
C05120=1225.014,-54.868,-38.670,179.937,5.334,148.946
C05121=1225.009,-54.618,-38.683,179.939,5.334,148.946
C05122=1225.004,-54.368,-38.695,179.941,5.334,148.945
C05123=1224.998,-54.118,-38.707,179.944,5.334,148.944
C05124=1224.993,-53.868,-38.719,179.947,5.335,148.944
C05125=1224.988,-53.619,-38.732,179.949,5.334,148.943
C05126=1224.983,-53.369,-38.743,179.952,5.335,148.942
C05127=1224.978,-53.120,-38.756,179.954,5.335,148.942
C05128=1224.973,-52.871,-38.768,179.956,5.335,148.941
C05129=1224.968,-52.621,-38.780,179.958,5.335,148.940
C05130=1224.963,-52.371,-38.793,179.961,5.335,148.939
C05131=1224.958,-52.121,-38.805,179.964,5.336,148.939
C05132=1224.952,-51.872,-38.817,179.966,5.335,148.938
C05133=1224.947,-51.622,-38.829,179.968,5.336,148.937
C05134=1224.942,-51.372,-38.842,179.971,5.335,148.937
C05135=1224.937,-51.123,-38.855,179.973,5.336,148.936
C05136=1224.931,-50.873,-38.866,179.976,5.336,148.935
C05137=1224.926,-50.624,-38.879,179.978,5.336,148.935
C05138=1224.921,-50.373,-38.891,179.981,5.337,148.934
C05139=1224.916,-50.124,-38.904,179.983,5.336,148.933
C05140=1224.911,-49.874,-38.916,179.985,5.337,148.932
C05141=1224.906,-49.624,-38.928,179.987,5.336,148.932
C05142=1224.901,-49.375,-38.941,179.990,5.337,148.931
C05143=1224.895,-49.126,-38.954,179.993,5.337,148.930
C05144=1224.890,-48.856,-38.967,179.995,5.337,148.930
C05145=1224.885,-48.586,-38.980,179.998,5.337,148.929
C05146=1224.880,-48.317,-38.994,-179.999,5.338,148.928
C05147=1224.874,-48.046,-39.007,-179.997,5.338,148.927
C05148=1224.868,-47.797,-39.020,-179.995,5.338,148.927
C05149=1224.863,-47.547,-39.032,-179.992,5.338,148.926
C05150=1224.858,-47.297,-39.045,-179.990,5.338,148.925
C05151=1224.853,-47.048,-39.057,-179.987,5.338,148.924
C05152=1224.848,-46.798,-39.070,-179.984,5.339,148.924
C05153=1224.843,-46.548,-39.082,-179.982,5.339,148.923
C05154=1224.838,-46.299,-39.094,-179.980,5.339,148.922
C05155=1224.833,-46.050,-39.107,-179.978,5.339,148.922
C05156=1224.828,-45.800,-39.120,-179.975,5.339,148.921
C05157=1224.823,-45.550,-39.132,-179.972,5.340,148.920
C05158=1224.817,-45.300,-39.144,-179.970,5.339,148.920
C05159=1224.812,-45.051,-39.157,-179.968,5.340,148.919
C05160=1224.807,-44.801,-39.170,-179.965,5.339,148.918
C05161=1224.802,-44.551,-39.183,-179.963,5.340,148.917
C05162=1224.796,-44.301,-39.195,-179.960,5.340,148.917
C05163=1224.791,-44.052,-39.208,-179.958,5.340,148.916
C05164=1224.786,-43.803,-39.220,-179.955,5.341,148.915
C05165=1224.782,-43.553,-39.233,-179.953,5.340,148.915
C05166=1224.777,-43.303,-39.246,-179.951,5.341,148.914
C05167=1224.771,-43.054,-39.258,-179.948,5.341,148.913
C05168=1224.766,-42.804,-39.270,-179.946,5.341,148.913
C05169=1224.761,-42.554,-39.284,-179.943,5.341,148.912
C05170=1224.756,-42.305,-39.296,-179.941,5.341,148.911
C05171=1224.751,-42.055,-39.309,-179.938,5.342,148.910
C05172=1224.745,-41.806,-39.322,-179.936,5.342,148.910
C05173=1224.741,-41.556,-39.335,-179.934,5.342,148.909
C05174=1224.736,-41.307,-39.347,-179.931,5.342,148.908
C05175=1224.730,-41.057,-39.359,-179.928,5.343,148.908
C05176=1224.725,-40.806,-39.373,-179.926,5.342,148.907
C05177=1224.720,-40.557,-39.385,-179.924,5.343,148.906
C05178=1224.715,-40.308,-39.398,-179.922,5.343,148.905
C05179=1224.710,-40.058,-39.410,-179.919,5.343,148.905
C05180=1224.705,-39.808,-39.423,-179.916,5.343,148.904
C05181=1224.699,-39.559,-39.437,-179.914,5.343,148.903
C05182=1224.694,-39.309,-39.449,-179.911,5.344,148.903
C05183=1224.690,-39.059,-39.462,-179.909,5.343,148.902
C05184=1224.685,-38.810,-39.475,-179.907,5.344,148.901
C05185=1224.679,-38.561,-39.487,-179.904,5.344,148.901
C05186=1224.674,-38.311,-39.501,-179.902,5.344,148.900
C05187=1224.669,-38.061,-39.513,-179.899,5.344,148.899
C05188=1224.664,-37.812,-39.526,-179.897,5.345,148.898
C05189=1224.659,-37.562,-39.539,-179.895,5.345,148.898
C05190=1224.654,-37.312,-39.552,-179.892,5.345,148.897
C05191=1224.648,-37.063,-39.565,-179.890,5.345,148.896
C05192=1224.643,-36.814,-39.577,-179.887,5.345,148.896
C05193=1224.639,-36.563,-39.590,-179.884,5.346,148.895
C05194=1224.633,-36.314,-39.604,-179.882,5.345,148.894
C05195=1224.628,-36.065,-39.616,-179.880,5.346,148.894
C05196=1224.623,-35.815,-39.629,-179.877,5.346,148.893
C05197=1224.618,-35.565,-39.642,-179.875,5.346,148.892
C05198=1224.612,-35.316,-39.655,-179.872,5.347,148.891
C05199=1224.608,-35.066,-39.668,-179.870,5.346,148.891
C05200=1224.603,-34.816,-39.681,-179.868,5.347,148.890
C05201=1224.597,-34.567,-39.694,-179.865,5.347,148.889
C05202=1224.592,-34.317,-39.707,-179.863,5.347,148.889
C05203=1224.587,-34.068,-39.720,-179.860,5.347,148.888
C05204=1224.582,-33.818,-39.734,-179.858,5.348,148.887
C05205=1224.577,-33.568,-39.746,-179.855,5.348,148.887
C05206=1224.572,-33.319,-39.759,-179.853,5.348,148.886
C05207=1224.567,-33.069,-39.772,-179.850,5.349,148.885
C05208=1224.562,-32.819,-39.785,-179.848,5.348,148.885
C05209=1224.556,-32.570,-39.798,-179.845,5.349,148.884
C05210=1224.551,-32.320,-39.811,-179.843,5.348,148.883
C05211=1224.546,-32.071,-39.824,-179.841,5.349,148.882
C05212=1224.542,-31.821,-39.837,-179.838,5.349,148.882
C05213=1224.536,-31.571,-39.851,-179.836,5.349,148.881
C05214=1224.531,-31.322,-39.863,-179.833,5.350,148.880
C05215=1224.526,-31.072,-39.876,-179.831,5.350,148.880
C05216=1224.520,-30.822,-39.889,-179.828,5.350,148.879
C05217=1224.516,-30.573,-39.903,-179.826,5.350,148.878
C05218=1224.510,-30.323,-39.916,-179.823,5.351,148.878
C05219=1224.506,-30.073,-39.929,-179.821,5.350,148.877
C05220=1224.501,-29.824,-39.942,-179.818,5.351,148.876
C05221=1224.495,-29.575,-39.956,-179.816,5.351,148.875
C05222=1224.491,-29.325,-39.969,-179.814,5.351,148.875
C05223=1224.485,-29.075,-39.982,-179.811,5.352,148.874
C05224=1224.480,-28.825,-39.995,-179.808,5.352,148.873
C05225=1224.475,-28.577,-40.008,-179.806,5.352,148.873
C05226=1224.470,-28.326,-40.022,-179.804,5.352,148.872
C05227=1224.465,-28.077,-40.034,-179.801,5.353,148.871
C05228=1224.460,-27.827,-40.048,-179.799,5.352,148.871
C05229=1224.455,-27.578,-40.061,-179.796,5.353,148.870
C05230=1224.449,-27.328,-40.074,-179.794,5.353,148.869
C05231=1224.445,-27.078,-40.087,-179.791,5.353,148.868
C05232=1224.439,-26.829,-40.101,-179.789,5.354,148.868
C05233=1224.435,-26.579,-40.114,-179.787,5.353,148.867
C05234=1224.429,-26.330,-40.127,-179.784,5.354,148.866
C05235=1224.424,-26.080,-40.141,-179.781,5.354,148.866
C05236=1224.419,-25.831,-40.154,-179.779,5.354,148.865
C05237=1224.414,-25.581,-40.167,-179.777,5.355,148.864
C05238=1224.409,-25.332,-40.181,-179.774,5.355,148.864
C05239=1224.404,-25.082,-40.194,-179.772,5.355,148.863
C05240=1224.399,-24.833,-40.207,-179.769,5.355,148.862
C05241=1224.394,-24.583,-40.221,-179.767,5.356,148.861
C05242=1224.388,-24.333,-40.234,-179.765,5.355,148.861
C05243=1224.384,-24.083,-40.248,-179.762,5.356,148.860
C05244=1224.378,-23.834,-40.261,-179.759,5.356,148.859
C05245=1224.374,-23.584,-40.275,-179.757,5.356,148.859
C05246=1224.368,-23.335,-40.288,-179.754,5.357,148.858
C05247=1224.363,-23.085,-40.301,-179.752,5.357,148.857
C05248=1224.358,-22.815,-40.316,-179.749,5.358,148.857
C05249=1224.352,-22.547,-40.331,-179.747,5.357,148.856
C05250=1224.347,-22.277,-40.344,-179.744,5.357,148.855
C05251=1224.341,-22.008,-40.359,-179.741,5.358,148.854
C05252=1224.336,-21.759,-40.373,-179.739,5.358,148.854
C05253=1224.331,-21.509,-40.386,-179.736,5.358,148.853
C05254=1224.326,-21.260,-40.400,-179.734,5.359,148.852
C05255=1224.321,-21.009,-40.413,-179.731,5.359,148.852
C05256=1224.316,-20.760,-40.427,-179.729,5.359,148.851
C05257=1224.310,-20.510,-40.440,-179.726,5.359,148.850
C05258=1224.306,-20.261,-40.454,-179.724,5.360,148.849
C05259=1224.300,-20.011,-40.467,-179.722,5.360,148.849
C05260=1224.296,-19.762,-40.481,-179.719,5.360,148.848
C05261=1224.290,-19.512,-40.494,-179.716,5.361,148.847
C05262=1224.285,-19.262,-40.508,-179.714,5.360,148.847
C05263=1224.281,-19.012,-40.521,-179.712,5.361,148.846
C05264=1224.275,-18.763,-40.535,-179.709,5.361,148.845
C05265=1224.270,-18.513,-40.549,-179.707,5.361,148.845
C05266=1224.265,-18.264,-40.562,-179.704,5.361,148.844
C05267=1224.260,-18.015,-40.577,-179.702,5.362,148.843
C05268=1224.254,-17.765,-40.590,-179.699,5.362,148.842
C05269=1224.250,-17.516,-40.603,-179.697,5.362,148.842
C05270=1224.245,-17.265,-40.617,-179.694,5.363,148.841
C05271=1224.239,-17.016,-40.631,-179.692,5.363,148.840
C05272=1224.235,-16.767,-40.645,-179.689,5.363,148.840
C05273=1224.230,-16.517,-40.658,-179.687,5.363,148.839
C05274=1224.224,-16.268,-40.672,-179.684,5.364,148.838
C05275=1224.220,-16.017,-40.685,-179.682,5.364,148.838
C05276=1224.214,-15.768,-40.699,-179.679,5.364,148.837
C05277=1224.209,-15.519,-40.713,-179.677,5.365,148.836
C05278=1224.204,-15.268,-40.727,-179.675,5.364,148.836
C05279=1224.199,-15.020,-40.740,-179.672,5.365,148.835
C05280=1224.194,-14.770,-40.754,-179.669,5.365,148.834
C05281=1224.189,-14.520,-40.768,-179.667,5.366,148.833
C05282=1224.184,-14.271,-40.781,-179.665,5.365,148.833
C05283=1224.179,-14.021,-40.795,-179.662,5.366,148.832
C05284=1224.174,-13.772,-40.810,-179.659,5.366,148.831
C05285=1224.168,-13.522,-40.823,-179.657,5.366,148.831
C05286=1224.164,-13.273,-40.837,-179.655,5.367,148.830
C05287=1224.159,-13.024,-40.851,-179.652,5.367,148.829
C05288=1224.154,-12.774,-40.865,-179.650,5.367,148.829
C05289=1224.148,-12.523,-40.878,-179.647,5.367,148.828
C05290=1224.143,-12.274,-40.893,-179.645,5.368,148.827
C05291=1224.139,-12.025,-40.906,-179.642,5.368,148.827
C05292=1224.134,-11.775,-40.920,-179.640,5.368,148.826
C05293=1224.128,-11.525,-40.934,-179.637,5.369,148.825
C05294=1224.123,-11.276,-40.948,-179.634,5.369,148.824
C05295=1224.119,-11.027,-40.961,-179.632,5.369,148.824
C05296=1224.114,-10.777,-40.976,-179.630,5.369,148.823
C05297=1224.108,-10.528,-40.990,-179.627,5.370,148.822
C05298=1224.103,-10.278,-41.003,-179.624,5.370,148.822
C05299=1224.098,-10.028,-41.017,-179.622,5.370,148.821
C05300=1224.092,-9.779,-41.031,-179.620,5.371,148.820
C05301=1224.088,-9.529,-41.045,-179.617,5.371,148.820
C05302=1224.083,-9.280,-41.059,-179.615,5.371,148.819
C05303=1224.078,-9.030,-41.074,-179.612,5.371,148.818
C05304=1224.072,-8.780,-41.087,-179.610,5.372,148.818
C05305=1224.067,-8.531,-41.101,-179.607,5.372,148.817
C05306=1224.062,-8.281,-41.115,-179.605,5.372,148.816
C05307=1224.058,-8.031,-41.130,-179.602,5.373,148.815
C05308=1224.053,-7.783,-41.143,-179.600,5.373,148.815
C05309=1224.048,-7.533,-41.157,-179.598,5.373,148.814
C05310=1224.043,-7.283,-41.172,-179.595,5.373,148.813
C05311=1224.038,-7.033,-41.186,-179.593,5.374,148.813
C05312=1224.032,-6.784,-41.200,-179.590,5.375,148.812
C05313=1224.027,-6.535,-41.214,-179.588,5.374,148.812
C05314=1224.022,-6.285,-41.228,-179.585,5.375,148.811
C05315=1224.017,-6.035,-41.243,-179.583,5.375,148.810
C05316=1224.012,-5.786,-41.256,-179.580,5.376,148.809
C05317=1224.007,-5.536,-41.269,-179.578,5.376,148.809
C05318=1224.002,-5.287,-41.284,-179.575,5.376,148.808
C05319=1223.997,-5.037,-41.298,-179.573,5.377,148.807
C05320=1223.992,-4.787,-41.312,-179.571,5.376,148.807
C05321=1223.987,-4.538,-41.326,-179.568,5.377,148.806
C05322=1223.982,-4.288,-41.340,-179.565,5.377,148.805
C05323=1223.977,-4.039,-41.355,-179.563,5.378,148.805
C05324=1223.972,-3.789,-41.369,-179.561,5.378,148.804
C05325=1223.966,-3.540,-41.383,-179.558,5.378,148.803
C05326=1223.962,-3.290,-41.397,-179.555,5.379,148.803
C05327=1223.957,-3.041,-41.411,-179.553,5.379,148.802
C05328=1223.952,-2.792,-41.426,-179.550,5.379,148.801
C05329=1223.947,-2.542,-41.441,-179.548,5.379,148.800
C05330=1223.942,-2.292,-41.455,-179.545,5.380,148.800
C05331=1223.936,-2.043,-41.469,-179.542,5.380,148.799
C05332=1223.932,-1.793,-41.483,-179.540,5.380,148.798
C05333=1223.927,-1.544,-41.497,-179.538,5.381,148.798
C05334=1223.922,-1.294,-41.512,-179.535,5.381,148.797
C05335=1223.917,-1.044,-41.526,-179.532,5.382,148.796
C05336=1223.912,-0.795,-41.540,-179.530,5.381,148.796
C05337=1223.906,-0.546,-41.554,-179.528,5.382,148.795
C05338=1223.901,-0.296,-41.568,-179.525,5.382,148.794
C05339=1223.897,-0.047,-41.583,-179.522,5.383,148.794
C05340=1223.892,0.203,-41.598,-179.520,5.383,148.793
C05341=1223.887,0.453,-41.612,-179.518,5.383,148.792
C05342=1223.882,0.702,-41.626,-179.515,5.384,148.792
C05343=1223.876,0.952,-41.641,-179.512,5.384,148.791
C05344=1223.870,1.201,-41.655,-179.510,5.384,148.790
C05345=1223.866,1.451,-41.670,-179.508,5.384,148.789
C05346=1223.861,1.700,-41.684,-179.505,5.385,148.789
C05347=1223.856,1.950,-41.699,-179.502,5.385,148.788
C05348=1223.851,2.200,-41.713,-179.500,5.385,148.787
C05349=1223.846,2.449,-41.727,-179.498,5.386,148.787
C05350=1223.841,2.698,-41.742,-179.495,5.386,148.786
C05351=1223.836,2.948,-41.756,-179.492,5.387,148.785
C05352=1223.831,3.216,-41.772,-179.490,5.387,148.785
C05353=1223.824,3.486,-41.787,-179.488,5.387,148.784
C05354=1223.819,3.755,-41.803,-179.485,5.387,148.783
C05355=1223.814,4.024,-41.819,-179.482,5.388,148.783
C05356=1223.809,4.273,-41.833,-179.480,5.389,148.782
C05357=1223.804,4.523,-41.847,-179.477,5.389,148.781
C05358=1223.799,4.772,-41.863,-179.474,5.390,148.781
C05359=1223.794,5.022,-41.877,-179.472,5.389,148.780
C05360=1223.789,5.272,-41.891,-179.470,5.390,148.779
C05361=1223.784,5.521,-41.906,-179.467,5.390,148.778
C05362=1223.779,5.771,-41.921,-179.464,5.391,148.778
C05363=1223.774,6.020,-41.935,-179.462,5.391,148.777
C05364=1223.769,6.270,-41.951,-179.460,5.391,148.776
C05365=1223.763,6.519,-41.965,-179.457,5.392,148.776
C05366=1223.759,6.768,-41.979,-179.454,5.392,148.775
C05367=1223.754,7.018,-41.994,-179.452,5.393,148.774
C05368=1223.749,7.267,-42.008,-179.450,5.392,148.774
C05369=1223.743,7.517,-42.023,-179.447,5.393,148.773
C05370=1223.739,7.766,-42.038,-179.444,5.393,148.772
C05371=1223.734,8.016,-42.052,-179.442,5.394,148.772
C05372=1223.729,8.265,-42.067,-179.440,5.394,148.771
C05373=1223.724,8.515,-42.081,-179.437,5.394,148.770
C05374=1223.718,8.765,-42.096,-179.434,5.395,148.770
C05375=1223.714,9.014,-42.111,-179.432,5.395,148.769
C05376=1223.709,9.264,-42.126,-179.429,5.396,148.768
C05377=1223.704,9.513,-42.141,-179.427,5.395,148.767
C05378=1223.698,9.763,-42.156,-179.424,5.396,148.767
C05379=1223.694,10.012,-42.170,-179.422,5.397,148.766
C05380=1223.689,10.262,-42.185,-179.419,5.397,148.766
C05381=1223.683,10.512,-42.200,-179.417,5.397,148.765
C05382=1223.678,10.761,-42.215,-179.415,5.398,148.764
C05383=1223.673,11.010,-42.229,-179.412,5.398,148.764
C05384=1223.669,11.260,-42.244,-179.409,5.399,148.763
C05385=1223.663,11.510,-42.259,-179.407,5.399,148.762
C05386=1223.659,11.759,-42.274,-179.405,5.399,148.762
C05387=1223.654,12.008,-42.288,-179.402,5.400,148.761
C05388=1223.648,12.258,-42.304,-179.399,5.400,148.760
C05389=1223.643,12.507,-42.318,-179.397,5.401,148.759
C05390=1223.639,12.757,-42.333,-179.394,5.401,148.759
C05391=1223.633,13.006,-42.348,-179.392,5.401,148.758
C05392=1223.628,13.256,-42.363,-179.389,5.401,148.757
C05393=1223.624,13.505,-42.378,-179.387,5.402,148.757
C05394=1223.618,13.756,-42.393,-179.384,5.402,148.756
C05395=1223.614,14.005,-42.408,-179.381,5.403,148.755
C05396=1223.609,14.254,-42.422,-179.379,5.403,148.755
C05397=1223.603,14.504,-42.438,-179.377,5.403,148.754
C05398=1223.599,14.753,-42.453,-179.374,5.404,148.753
C05399=1223.593,15.003,-42.468,-179.371,5.404,148.753
C05400=1223.588,15.252,-42.483,-179.369,5.405,148.752
C05401=1223.584,15.502,-42.497,-179.367,5.406,148.752
C05402=1223.578,15.751,-42.513,-179.364,5.405,148.751
C05403=1223.574,16.000,-42.528,-179.362,5.406,148.750
C05404=1223.568,16.250,-42.542,-179.359,5.406,148.749
C05405=1223.563,16.499,-42.557,-179.357,5.407,148.749
C05406=1223.559,16.748,-42.572,-179.354,5.408,148.748
C05407=1223.553,16.999,-42.588,-179.352,5.407,148.747
C05408=1223.549,17.248,-42.603,-179.349,5.408,148.747
C05409=1223.543,17.498,-42.618,-179.347,5.408,148.746
C05410=1223.538,17.747,-42.633,-179.344,5.409,148.745
C05411=1223.533,17.997,-42.648,-179.341,5.409,148.745
C05412=1223.528,18.246,-42.663,-179.339,5.409,148.744
C05413=1223.524,18.495,-42.678,-179.336,5.410,148.743
C05414=1223.518,18.745,-42.693,-179.334,5.410,148.743
C05415=1223.513,18.994,-42.708,-179.331,5.411,148.742
C05416=1223.509,19.244,-42.724,-179.329,5.411,148.741
C05417=1223.504,19.494,-42.738,-179.326,5.412,148.741
C05418=1223.498,19.743,-42.754,-179.324,5.412,148.740
C05419=1223.494,19.992,-42.769,-179.322,5.412,148.739
C05420=1223.488,20.242,-42.784,-179.319,5.413,148.739
C05421=1223.484,20.491,-42.799,-179.316,5.414,148.738
C05422=1223.478,20.741,-42.814,-179.314,5.414,148.737
C05423=1223.474,20.991,-42.830,-179.311,5.415,148.737
C05424=1223.468,21.240,-42.845,-179.309,5.414,148.736
C05425=1223.464,21.489,-42.860,-179.306,5.415,148.735
C05426=1223.458,21.738,-42.876,-179.304,5.415,148.735
C05427=1223.453,21.988,-42.890,-179.301,5.416,148.734
C05428=1223.448,22.238,-42.906,-179.298,5.416,148.733
C05429=1223.443,22.488,-42.922,-179.296,5.417,148.733
C05430=1223.439,22.737,-42.937,-179.294,5.417,148.732
C05431=1223.433,22.986,-42.952,-179.291,5.417,148.731
C05432=1223.429,23.235,-42.967,-179.288,5.418,148.731
C05433=1223.423,23.485,-42.983,-179.286,5.419,148.730
C05434=1223.419,23.734,-42.998,-179.284,5.419,148.729
C05435=1223.413,23.984,-43.013,-179.281,5.420,148.729
C05436=1223.408,24.234,-43.029,-179.278,5.420,148.728
C05437=1223.403,24.483,-43.044,-179.276,5.420,148.727
C05438=1223.398,24.732,-43.059,-179.274,5.421,148.727
C05439=1223.394,24.982,-43.075,-179.271,5.421,148.726
C05440=1223.389,25.232,-43.090,-179.268,5.422,148.725
C05441=1223.383,25.481,-43.106,-179.266,5.422,148.725
C05442=1223.379,25.730,-43.121,-179.263,5.423,148.724
C05443=1223.374,25.980,-43.137,-179.261,5.422,148.723
C05444=1223.369,26.229,-43.152,-179.258,5.423,148.723
C05445=1223.364,26.479,-43.167,-179.256,5.424,148.722
C05446=1223.358,26.728,-43.183,-179.254,5.424,148.722
C05447=1223.354,26.978,-43.198,-179.251,5.425,148.721
C05448=1223.349,27.227,-43.214,-179.248,5.426,148.720
C05449=1223.344,27.477,-43.229,-179.246,5.426,148.719
C05450=1223.339,27.726,-43.244,-179.244,5.426,148.719
C05451=1223.334,27.976,-43.260,-179.241,5.426,148.718
C05452=1223.329,28.225,-43.276,-179.238,5.427,148.717
C05453=1223.324,28.474,-43.291,-179.236,5.427,148.717
C05454=1223.319,28.724,-43.306,-179.233,5.428,148.716
C05455=1223.314,28.974,-43.322,-179.230,5.429,148.715
C05456=1223.308,29.242,-43.339,-179.228,5.429,148.715
C05457=1223.304,29.510,-43.356,-179.225,5.430,148.714
C05458=1223.298,29.780,-43.372,-179.222,5.430,148.713
C05459=1223.292,30.048,-43.389,-179.220,5.431,148.713
C05460=1223.287,30.298,-43.405,-179.217,5.431,148.712
C05461=1223.283,30.547,-43.420,-179.214,5.432,148.711
C05462=1223.278,30.796,-43.436,-179.212,5.432,148.711
C05463=1223.272,31.045,-43.452,-179.210,5.432,148.710
C05464=1223.267,31.296,-43.468,-179.207,5.433,148.709
C05465=1223.263,31.545,-43.483,-179.204,5.433,148.709
C05466=1223.257,31.794,-43.499,-179.202,5.434,148.708
C05467=1223.253,32.044,-43.514,-179.199,5.434,148.707
C05468=1223.247,32.294,-43.530,-179.197,5.435,148.707
C05469=1223.243,32.542,-43.546,-179.194,5.436,148.706
C05470=1223.238,32.792,-43.562,-179.192,5.435,148.705
C05471=1223.233,33.042,-43.577,-179.190,5.436,148.705
C05472=1223.227,33.291,-43.593,-179.187,5.437,148.704
C05473=1223.223,33.541,-43.609,-179.184,5.437,148.703
C05474=1223.218,33.790,-43.625,-179.182,5.438,148.703
C05475=1223.213,34.039,-43.640,-179.179,5.438,148.702
C05476=1223.208,34.289,-43.656,-179.176,5.439,148.701
C05477=1223.203,34.538,-43.672,-179.174,5.439,148.701
C05478=1223.198,34.788,-43.688,-179.172,5.440,148.700
C05479=1223.193,35.037,-43.704,-179.170,5.440,148.700
C05480=1223.188,35.286,-43.719,-179.167,5.440,148.699
C05481=1223.183,35.537,-43.735,-179.164,5.441,148.698
